  MoveL 3161 to (509.6, 500.88, 6.4) mm, rotated rx 0 ry 90 rz 0 deg; joints [-11.904, -26.782, 109.906, -15.94, -82.523, 51.112]
  Call Extruder(0.254)
  MoveL 3162 to (509.6, 509.6, 6.4) mm, rotated rx 0 ry 90 rz 0 deg; joints [-12.688, -26.745, 109.678, -16.738, -82.366, 51.259]
  Call Extruder(0.559)
  MoveL 3163 to (490.4, 509.6, 6.4) mm, rotated rx 0 ry 90 rz 0 deg; joints [-13.088, -27.092, 111.961, -17.074, -84.231, 50.733]
  MoveL 3164 to (490.4, 490.4, 6.4) mm, rotated rx 0 ry 90 rz 0 deg; joints [-11.303, -27.159, 112.45, -15.27, -84.594, 50.467]
  Call Extruder(0.167)
  MoveL 3165 to (496.12, 490.4, 6.4) mm, rotated rx 0 ry 90 rz 0 deg; joints [-11.197, -27.066, 111.773, -15.179, -84.029, 50.612]
  Call Extruder(0.055)
  MoveL 3166 to (496.12, 492.3, 6.4) mm, rotated rx 0 ry 90 rz 0 deg; joints [-11.373, -27.06, 111.728, -15.356, -83.995, 50.638]
  Call Extruder(0.073)
  MoveL 3167 to (498.63, 492.29, 6.4) mm, rotated rx 0 ry 90 rz 0 deg; joints [-11.326, -27.017, 111.43, -15.316, -83.748, 50.702]
  Call Extruder(0.045)
  MoveL 3168 to (498.63, 490.75, 6.4) mm, rotated rx 0 ry 90 rz 0 deg; joints [-11.183, -27.022, 111.466, -15.172, -83.775, 50.68]
  Call Extruder(0.010)
  MoveL 3169 to (498.63, 490.4, 6.4) mm, rotated rx 0 ry 90 rz 0 deg; joints [-11.151, -27.023, 111.474, -15.14, -83.781, 50.675]
  Call Extruder(0.007)
  MoveL 3170 to (498.98, 490.4, 6.4) mm, rotated rx 0 ry 90 rz 0 deg; joints [-11.145, -27.017, 111.433, -15.134, -83.746, 50.684]
  Call Extruder(0.044)
  MoveL 3171 to (500.51, 490.4, 6.4) mm, rotated rx 0 ry 90 rz 0 deg; joints [-11.117, -26.99, 111.251, -15.111, -83.596, 50.722]
  Call Extruder(0.045)
  MoveL 3172 to (500.51, 491.94, 6.4) mm, rotated rx 0 ry 90 rz 0 deg; joints [-11.259, -26.985, 111.215, -15.255, -83.569, 50.744]
  Call Extruder(0.010)
  MoveL 3173 to (500.51, 492.29, 6.4) mm, rotated rx 0 ry 90 rz 0 deg; joints [-11.291, -26.984, 111.207, -15.287, -83.563, 50.749]
  Call Extruder(0.007)
  MoveL 3174 to (500.86, 492.29, 6.4) mm, rotated rx 0 ry 90 rz 0 deg; joints [-11.285, -26.978, 111.165, -15.282, -83.529, 50.758]
  Call Extruder(0.063)
  MoveL 3175 to (503.03, 492.3, 6.4) mm, rotated rx 0 ry 90 rz 0 deg; joints [-11.245, -26.939, 110.906, -15.249, -83.315, 50.812]
  Call Extruder(0.055)
  MoveL 3176 to (503.03, 490.4, 6.4) mm, rotated rx 0 ry 90 rz 0 deg; joints [-11.072, -26.946, 110.95, -15.073, -83.347, 50.785]
  Call Extruder(0.191)
  MoveL 3177 to (509.6, 490.4, 6.4) mm, rotated rx 0 ry 90 rz 0 deg; joints [-10.955, -26.823, 110.161, -14.976, -82.7, 50.946]
  Call Extruder(0.233)
  MoveL 3178 to (509.6, 498.4, 6.4) mm, rotated rx 0 ry 90 rz 0 deg; joints [-11.68, -26.793, 109.969, -15.712, -82.566, 51.072]
  Call Extruder(0.056)
  MoveL 3179 to (507.66, 498.4, 6.4) mm, rotated rx 0 ry 90 rz 0 deg; joints [-11.716, -26.83, 110.202, -15.742, -82.756, 51.023]
  Set speed (120.0 mm/s)
  MoveL 3180 to (507.66, 498.8, 6.4) mm, rotated rx 0 ry 90 rz 0 deg; joints [-11.752, -26.828, 110.192, -15.779, -82.749, 51.029]
  Set speed (1000.0 mm/s)
  MoveL 3181 to (506.96, 498.8, 6.4) mm, rotated rx 0 ry 90 rz 0 deg; joints [-11.766, -26.842, 110.276, -15.79, -82.818, 51.011]
  Set speed (1000.0 mm/s)
  MoveL 3182 to (490.68, 490.68, 6.4) mm, rotated rx 0 ry 90 rz 0 deg; joints [-11.324, -27.154, 112.411, -15.292, -84.562, 50.478]
  Set speed (1000.0 mm/s)
  MoveL 3183 to (490.68, 490.68, 6.5) mm, rotated rx 0 ry 90 rz 0 deg; joints [-11.324, -27.165, 112.416, -15.292, -84.557, 50.479]
  Set speed (30.0 mm/s)
  Call Extruder(0.767)
  MoveL 3184 to (509.32, 509.32, 6.5) mm, rotated rx 0 ry 90 rz 0 deg; joints [-12.669, -26.762, 109.724, -16.717, -82.394, 51.248]
  MoveL 3185 to (509.44, 509.44, 6.5) mm, rotated rx 0 ry 90 rz 0 deg; joints [-12.677, -26.76, 109.706, -16.726, -82.38, 51.253]
  Set speed (120.0 mm/s)
  MoveL 3186 to (508.74, 501.16, 6.5) mm, rotated rx 0 ry 90 rz 0 deg; joints [-11.945, -26.809, 110.008, -15.979, -82.598, 51.096]
  Set speed (30.0 mm/s)
  Call Extruder(0.336)
  MoveL 3187 to (500.58, 509.32, 6.5) mm, rotated rx 0 ry 90 rz 0 deg; joints [-12.847, -26.928, 110.77, -16.865, -83.242, 51.012]
  Set speed (120.0 mm/s)
  MoveL 3188 to (499.42, 509.32, 6.5) mm, rotated rx 0 ry 90 rz 0 deg; joints [-12.872, -26.949, 110.907, -16.885, -83.355, 50.98]
  Set speed (30.0 mm/s)
  Call Extruder(0.360)
  MoveL 3189 to (490.68, 500.58, 6.5) mm, rotated rx 0 ry 90 rz 0 deg; joints [-12.247, -27.132, 112.172, -16.224, -84.375, 50.612]
  Set speed (120.0 mm/s)
  MoveL 3190 to (490.68, 499.42, 6.5) mm, rotated rx 0 ry 90 rz 0 deg; joints [-12.139, -27.136, 112.202, -16.115, -84.397, 50.596]
  Set speed (30.0 mm/s)
  Call Extruder(0.282)
  MoveL 3191 to (497.52, 492.57, 6.5) mm, rotated rx 0 ry 90 rz 0 deg; joints [-11.372, -27.045, 111.56, -15.36, -83.847, 50.679]
  MoveL 3192 to (497.65, 492.45, 6.5) mm, rotated rx 0 ry 90 rz 0 deg; joints [-11.359, -27.044, 111.549, -15.347, -83.837, 50.68]
  Set speed (120.0 mm/s)
  MoveL 3193 to (498.97, 491.13, 6.5) mm, rotated rx 0 ry 90 rz 0 deg; joints [-11.212, -27.025, 111.422, -15.202, -83.73, 50.695]
  Set speed (30.0 mm/s)
  Call Extruder(0.018)
  MoveL 3194 to (499.42, 490.68, 6.5) mm, rotated rx 0 ry 90 rz 0 deg; joints [-11.163, -27.019, 111.38, -15.154, -83.693, 50.7]
  Set speed (120.0 mm/s)
  MoveL 3195 to (500.42, 492.32, 6.5) mm, rotated rx 0 ry 90 rz 0 deg; joints [-11.296, -26.996, 111.222, -15.292, -83.567, 50.749]
  Set speed (1000.0 mm/s)
  MoveL 3196 to (502.47, 492.57, 6.5) mm, rotated rx 0 ry 90 rz 0 deg; joints [-11.281, -26.958, 110.97, -15.283, -83.36, 50.804]
  Set speed (30.0 mm/s)
  Call Extruder(0.228)
  MoveL 3197 to (508.02, 498.12, 6.5) mm, rotated rx 0 ry 90 rz 0 deg; joints [-11.684, -26.835, 110.171, -15.711, -82.721, 51.029]
  MoveL 3198 to (508.14, 498.24, 6.5) mm, rotated rx 0 ry 90 rz 0 deg; joints [-11.693, -26.832, 110.153, -15.72, -82.707, 51.034]
  Set speed (120.0 mm/s)
  MoveL 3199 to (509.32, 490.68, 6.5) mm, rotated rx 0 ry 90 rz 0 deg; joints [-10.985, -26.838, 110.194, -15.006, -82.718, 50.945]
  Set speed (30.0 mm/s)
  Call Extruder(0.767)
  MoveL 3200 to (490.68, 509.32, 6.5) mm, rotated rx 0 ry 90 rz 0 deg; joints [-13.056, -27.1, 111.941, -17.043, -84.205, 50.738]
  MoveL 3201 to (490.56, 509.44, 6.5) mm, rotated rx 0 ry 90 rz 0 deg; joints [-13.07, -27.101, 111.952, -17.057, -84.214, 50.736]
  Set speed (120.0 mm/s)
  MoveL 3202 to (507.59, 498.33, 6.5) mm, rotated rx 0 ry 90 rz 0 deg; joints [-11.711, -26.842, 110.217, -15.737, -82.759, 51.021]
  Set speed (1000.0 mm/s)
  MoveL 3203 to (507.66, 498.4, 6.5) mm, rotated rx 0 ry 90 rz 0 deg; joints [-11.716, -26.84, 110.207, -15.742, -82.751, 51.024]
  Set speed (15.0 mm/s)
  Call Extruder(0.072)
  MoveL 3204 to (507.66, 500.88, 6.5) mm, rotated rx 0 ry 90 rz 0 deg; joints [-11.941, -26.83, 110.145, -15.97, -82.708, 51.064]
  Call Extruder(0.056)
  MoveL 3205 to (509.6, 500.88, 6.5) mm, rotated rx 0 ry 90 rz 0 deg; joints [-11.904, -26.793, 109.911, -15.94, -82.518, 51.114]
  Call Extruder(0.254)
  MoveL 3206 to (509.6, 509.6, 6.5) mm, rotated rx 0 ry 90 rz 0 deg; joints [-12.688, -26.756, 109.683, -16.738, -82.361, 51.26]
  Call Extruder(0.559)
  MoveL 3207 to (490.4, 509.6, 6.5) mm, rotated rx 0 ry 90 rz 0 deg; joints [-13.088, -27.103, 111.966, -17.074, -84.226, 50.734]
  MoveL 3208 to (490.4, 490.4, 6.5) mm, rotated rx 0 ry 90 rz 0 deg; joints [-11.303, -27.17, 112.456, -15.27, -84.589, 50.468]
  Call Extruder(0.168)
  MoveL 3209 to (496.18, 490.4, 6.5) mm, rotated rx 0 ry 90 rz 0 deg; joints [-11.196, -27.076, 111.772, -15.178, -84.018, 50.615]
  Call Extruder(0.045)
  MoveL 3210 to (496.18, 491.94, 6.5) mm, rotated rx 0 ry 90 rz 0 deg; joints [-11.339, -27.07, 111.735, -15.323, -83.991, 50.636]
  Call Extruder(0.010)
  MoveL 3211 to (496.18, 492.3, 6.5) mm, rotated rx 0 ry 90 rz 0 deg; joints [-11.372, -27.069, 111.727, -15.355, -83.985, 50.641]
  Call Extruder(0.007)
  MoveL 3212 to (496.53, 492.3, 6.5) mm, rotated rx 0 ry 90 rz 0 deg; joints [-11.365, -27.063, 111.685, -15.35, -83.95, 50.65]
  Call Extruder(0.063)
  MoveL 3213 to (498.69, 492.29, 6.5) mm, rotated rx 0 ry 90 rz 0 deg; joints [-11.325, -27.026, 111.428, -15.316, -83.737, 50.705]
  Call Extruder(0.045)
  MoveL 3214 to (498.69, 490.75, 6.5) mm, rotated rx 0 ry 90 rz 0 deg; joints [-11.182, -27.032, 111.465, -15.172, -83.764, 50.683]
  Call Extruder(0.010)
  MoveL 3215 to (498.69, 490.4, 6.5) mm, rotated rx 0 ry 90 rz 0 deg; joints [-11.15, -27.033, 111.473, -15.139, -83.77, 50.678]
  Call Extruder(0.007)
  MoveL 3216 to (499.04, 490.4, 6.5) mm, rotated rx 0 ry 90 rz 0 deg; joints [-11.144, -27.027, 111.431, -15.133, -83.735, 50.687]
  Call Extruder(0.041)
  MoveL 3217 to (500.45, 490.4, 6.5) mm, rotated rx 0 ry 90 rz 0 deg; joints [-11.118, -27.002, 111.264, -15.112, -83.597, 50.722]
  Call Extruder(0.045)
  MoveL 3218 to (500.45, 491.94, 6.5) mm, rotated rx 0 ry 90 rz 0 deg; joints [-11.26, -26.997, 111.227, -15.256, -83.57, 50.744]
  Call Extruder(0.010)
  MoveL 3219 to (500.45, 492.29, 6.5) mm, rotated rx 0 ry 90 rz 0 deg; joints [-11.293, -26.996, 111.219, -15.288, -83.564, 50.749]
  Call Extruder(0.007)
  MoveL 3220 to (500.8, 492.29, 6.5) mm, rotated rx 0 ry 90 rz 0 deg; joints [-11.286, -26.989, 111.177, -15.283, -83.53, 50.758]
  Call Extruder(0.063)
  MoveL 3221 to (502.96, 492.3, 6.5) mm, rotated rx 0 ry 90 rz 0 deg; joints [-11.247, -26.951, 110.918, -15.25, -83.316, 50.812]
  Call Extruder(0.055)
  MoveL 3222 to (502.97, 490.4, 6.5) mm, rotated rx 0 ry 90 rz 0 deg; joints [-11.073, -26.957, 110.963, -15.074, -83.348, 50.784]
  Call Extruder(0.193)
  MoveL 3223 to (509.6, 490.4, 6.5) mm, rotated rx 0 ry 90 rz 0 deg; joints [-10.955, -26.834, 110.167, -14.977, -82.695, 50.948]
  Call Extruder(0.233)
  MoveL 3224 to (509.6, 498.4, 6.5) mm, rotated rx 0 ry 90 rz 0 deg; joints [-11.68, -26.803, 109.974, -15.712, -82.561, 51.074]
  Call Extruder(0.056)
  MoveL 3225 to (507.66, 498.4, 6.5) mm, rotated rx 0 ry 90 rz 0 deg; joints [-11.716, -26.84, 110.207, -15.742, -82.751, 51.024]
  Set speed (120.0 mm/s)
  MoveL 3226 to (507.66, 498.8, 6.5) mm, rotated rx 0 ry 90 rz 0 deg; joints [-11.752, -26.839, 110.197, -15.779, -82.744, 51.03]
  Set speed (1000.0 mm/s)
  MoveL 3227 to (506.96, 498.8, 6.5) mm, rotated rx 0 ry 90 rz 0 deg; joints [-11.766, -26.852, 110.281, -15.79, -82.813, 51.013]
  Set speed (1000.0 mm/s)
  MoveL 3228 to (490.68, 490.68, 6.5) mm, rotated rx 0 ry 90 rz 0 deg; joints [-11.324, -27.165, 112.416, -15.292, -84.557, 50.479]
  Set speed (1000.0 mm/s)
  MoveL 3229 to (490.68, 490.68, 6.6) mm, rotated rx 0 ry 90 rz 0 deg; joints [-11.324, -27.175, 112.421, -15.292, -84.551, 50.481]
  Set speed (30.0 mm/s)
  Call Extruder(0.767)
  MoveL 3230 to (509.32, 509.32, 6.6) mm, rotated rx 0 ry 90 rz 0 deg; joints [-12.669, -26.773, 109.729, -16.717, -82.389, 51.25]
  MoveL 3231 to (509.44, 509.44, 6.6) mm, rotated rx 0 ry 90 rz 0 deg; joints [-12.677, -26.77, 109.711, -16.726, -82.375, 51.255]
  Set speed (120.0 mm/s)
  MoveL 3232 to (508.74, 501.16, 6.6) mm, rotated rx 0 ry 90 rz 0 deg; joints [-11.945, -26.819, 110.013, -15.979, -82.592, 51.098]
  Set speed (30.0 mm/s)
  Call Extruder(0.336)
  MoveL 3233 to (500.58, 509.32, 6.6) mm, rotated rx 0 ry 90 rz 0 deg; joints [-12.847, -26.938, 110.775, -16.865, -83.237, 51.013]
  Set speed (120.0 mm/s)
  MoveL 3234 to (499.42, 509.32, 6.6) mm, rotated rx 0 ry 90 rz 0 deg; joints [-12.872, -26.959, 110.913, -16.886, -83.35, 50.982]
  Set speed (30.0 mm/s)
  Call Extruder(0.360)
  MoveL 3235 to (490.68, 500.58, 6.6) mm, rotated rx 0 ry 90 rz 0 deg; joints [-12.247, -27.142, 112.178, -16.224, -84.37, 50.614]
  Set speed (120.0 mm/s)
  MoveL 3236 to (490.68, 499.42, 6.6) mm, rotated rx 0 ry 90 rz 0 deg; joints [-12.139, -27.146, 112.207, -16.115, -84.392, 50.598]
  Set speed (30.0 mm/s)
  Call Extruder(0.282)
  MoveL 3237 to (497.52, 492.57, 6.6) mm, rotated rx 0 ry 90 rz 0 deg; joints [-11.372, -27.056, 111.566, -15.36, -83.842, 50.68]
  MoveL 3238 to (497.65, 492.45, 6.6) mm, rotated rx 0 ry 90 rz 0 deg; joints [-11.359, -27.054, 111.554, -15.347, -83.832, 50.682]
  Set speed (120.0 mm/s)
  MoveL 3239 to (499.03, 491.07, 6.6) mm, rotated rx 0 ry 90 rz 0 deg; joints [-11.205, -27.035, 111.422, -15.196, -83.72, 50.697]
  Set speed (30.0 mm/s)
  Call Extruder(0.016)
  MoveL 3240 to (499.42, 490.68, 6.6) mm, rotated rx 0 ry 90 rz 0 deg; joints [-11.163, -27.03, 111.385, -15.154, -83.688, 50.702]
  Set speed (120.0 mm/s)
  MoveL 3241 to (500.36, 492.32, 6.6) mm, rotated rx 0 ry 90 rz 0 deg; joints [-11.297, -27.008, 111.234, -15.293, -83.568, 50.748]
  Set speed (1000.0 mm/s)
  MoveL 3242 to (502.47, 492.57, 6.6) mm, rotated rx 0 ry 90 rz 0 deg; joints [-11.281, -26.969, 110.976, -15.284, -83.355, 50.805]
  Set speed (30.0 mm/s)
  Call Extruder(0.228)
  MoveL 3243 to (508.02, 498.12, 6.6) mm, rotated rx 0 ry 90 rz 0 deg; joints [-11.684, -26.845, 110.176, -15.711, -82.716, 51.03]
  MoveL 3244 to (508.14, 498.24, 6.6) mm, rotated rx 0 ry 90 rz 0 deg; joints [-11.693, -26.842, 110.159, -15.72, -82.702, 51.035]
  Set speed (120.0 mm/s)
  MoveL 3245 to (509.32, 490.68, 6.6) mm, rotated rx 0 ry 90 rz 0 deg; joints [-10.985, -26.849, 110.199, -15.006, -82.713, 50.946]
  Set speed (30.0 mm/s)
  Call Extruder(0.767)
  MoveL 3246 to (490.68, 509.32, 6.6) mm, rotated rx 0 ry 90 rz 0 deg; joints [-13.056, -27.11, 111.947, -17.043, -84.2, 50.74]
  MoveL 3247 to (490.56, 509.44, 6.6) mm, rotated rx 0 ry 90 rz 0 deg; joints [-13.07, -27.112, 111.958, -17.057, -84.209, 50.738]
  Set speed (120.0 mm/s)
  MoveL 3248 to (507.59, 498.33, 6.6) mm, rotated rx 0 ry 90 rz 0 deg; joints [-11.711, -26.852, 110.223, -15.737, -82.754, 51.023]
  Set speed (1000.0 mm/s)
  MoveL 3249 to (507.66, 498.4, 6.6) mm, rotated rx 0 ry 90 rz 0 deg; joints [-11.716, -26.851, 110.212, -15.742, -82.746, 51.026]
  Set speed (15.0 mm/s)
  Call Extruder(0.072)
  MoveL 3250 to (507.66, 500.88, 6.6) mm, rotated rx 0 ry 90 rz 0 deg; joints [-11.941, -26.841, 110.15, -15.97, -82.703, 51.065]
  Call Extruder(0.056)
  MoveL 3251 to (509.6, 500.88, 6.6) mm, rotated rx 0 ry 90 rz 0 deg; joints [-11.904, -26.803, 109.917, -15.94, -82.513, 51.115]
  Call Extruder(0.254)
  MoveL 3252 to (509.6, 509.6, 6.6) mm, rotated rx 0 ry 90 rz 0 deg; joints [-12.688, -26.766, 109.688, -16.738, -82.356, 51.262]
  Call Extruder(0.559)
  MoveL 3253 to (490.4, 509.6, 6.6) mm, rotated rx 0 ry 90 rz 0 deg; joints [-13.088, -27.114, 111.972, -17.074, -84.221, 50.736]
  MoveL 3254 to (490.4, 490.4, 6.6) mm, rotated rx 0 ry 90 rz 0 deg; joints [-11.303, -27.181, 112.461, -15.27, -84.584, 50.47]
  Call Extruder(0.170)
  MoveL 3255 to (496.23, 490.4, 6.6) mm, rotated rx 0 ry 90 rz 0 deg; joints [-11.195, -27.085, 111.771, -15.177, -84.007, 50.618]
  Call Extruder(0.055)
  MoveL 3256 to (496.24, 492.3, 6.6) mm, rotated rx 0 ry 90 rz 0 deg; joints [-11.371, -27.079, 111.725, -15.355, -83.974, 50.644]
  Call Extruder(0.073)
  MoveL 3257 to (498.75, 492.29, 6.6) mm, rotated rx 0 ry 90 rz 0 deg; joints [-11.324, -27.036, 111.426, -15.315, -83.726, 50.708]
  Call Extruder(0.045)
  MoveL 3258 to (498.75, 490.75, 6.6) mm, rotated rx 0 ry 90 rz 0 deg; joints [-11.181, -27.041, 111.463, -15.171, -83.753, 50.686]
  Call Extruder(0.010)
  MoveL 3259 to (498.75, 490.4, 6.6) mm, rotated rx 0 ry 90 rz 0 deg; joints [-11.149, -27.042, 111.471, -15.138, -83.759, 50.681]
  Call Extruder(0.007)
  MoveL 3260 to (499.1, 490.4, 6.6) mm, rotated rx 0 ry 90 rz 0 deg; joints [-11.143, -27.036, 111.429, -15.133, -83.724, 50.69]
  Call Extruder(0.037)
  MoveL 3261 to (500.39, 490.4, 6.6) mm, rotated rx 0 ry 90 rz 0 deg; joints [-11.119, -27.014, 111.276, -15.113, -83.597, 50.722]
  Call Extruder(0.045)
  MoveL 3262 to (500.38, 491.94, 6.6) mm, rotated rx 0 ry 90 rz 0 deg; joints [-11.261, -27.008, 111.24, -15.257, -83.571, 50.744]
  Call Extruder(0.010)
  MoveL 3263 to (500.39, 492.29, 6.6) mm, rotated rx 0 ry 90 rz 0 deg; joints [-11.294, -27.007, 111.232, -15.29, -83.565, 50.749]
  Call Extruder(0.007)
  MoveL 3264 to (500.73, 492.29, 6.6) mm, rotated rx 0 ry 90 rz 0 deg; joints [-11.287, -27.001, 111.19, -15.284, -83.531, 50.758]
  Call Extruder(0.063)
  MoveL 3265 to (502.9, 492.3, 6.6) mm, rotated rx 0 ry 90 rz 0 deg; joints [-11.248, -26.962, 110.931, -15.251, -83.318, 50.812]
  Call Extruder(0.055)
  MoveL 3266 to (502.9, 490.4, 6.6) mm, rotated rx 0 ry 90 rz 0 deg; joints [-11.074, -26.969, 110.976, -15.075, -83.349, 50.784]
  Call Extruder(0.195)
  MoveL 3267 to (509.6, 490.4, 6.6) mm, rotated rx 0 ry 90 rz 0 deg; joints [-10.955, -26.844, 110.172, -14.977, -82.69, 50.949]
  Call Extruder(0.233)
  MoveL 3268 to (509.6, 498.4, 6.6) mm, rotated rx 0 ry 90 rz 0 deg; joints [-11.68, -26.813, 109.979, -15.713, -82.556, 51.075]
  Call Extruder(0.056)
  MoveL 3269 to (507.66, 498.4, 6.6) mm, rotated rx 0 ry 90 rz 0 deg; joints [-11.716, -26.851, 110.212, -15.742, -82.746, 51.026]
  Set speed (120.0 mm/s)
  MoveL 3270 to (507.66, 498.8, 6.6) mm, rotated rx 0 ry 90 rz 0 deg; joints [-11.752, -26.849, 110.202, -15.779, -82.739, 51.032]
  Set speed (1000.0 mm/s)
  MoveL 3271 to (506.96, 498.8, 6.6) mm, rotated rx 0 ry 90 rz 0 deg; joints [-11.765, -26.863, 110.287, -15.79, -82.808, 51.014]
  Set speed (1000.0 mm/s)
  MoveL 3272 to (490.68, 490.68, 6.6) mm, rotated rx 0 ry 90 rz 0 deg; joints [-11.324, -27.175, 112.421, -15.292, -84.551, 50.481]
  Set speed (1000.0 mm/s)
  MoveL 3273 to (490.68, 490.68, 6.7) mm, rotated rx 0 ry 90 rz 0 deg; joints [-11.324, -27.186, 112.427, -15.292, -84.546, 50.482]
  Set speed (30.0 mm/s)
  Call Extruder(0.767)
  MoveL 3274 to (509.32, 509.32, 6.7) mm, rotated rx 0 ry 90 rz 0 deg; joints [-12.669, -26.783, 109.735, -16.717, -82.384, 51.251]
  MoveL 3275 to (509.44, 509.44, 6.7) mm, rotated rx 0 ry 90 rz 0 deg; joints [-12.677, -26.78, 109.717, -16.727, -82.37, 51.257]
  Set speed (120.0 mm/s)
  MoveL 3276 to (508.74, 501.16, 6.7) mm, rotated rx 0 ry 90 rz 0 deg; joints [-11.945, -26.829, 110.018, -15.979, -82.587, 51.099]
  Set speed (30.0 mm/s)
  Call Extruder(0.336)
  MoveL 3277 to (500.58, 509.32, 6.7) mm, rotated rx 0 ry 90 rz 0 deg; joints [-12.847, -26.949, 110.78, -16.866, -83.232, 51.015]
  Set speed (120.0 mm/s)
  MoveL 3278 to (499.42, 509.32, 6.7) mm, rotated rx 0 ry 90 rz 0 deg; joints [-12.872, -26.97, 110.918, -16.886, -83.345, 50.983]
  Set speed (30.0 mm/s)
  Call Extruder(0.360)
  MoveL 3279 to (490.68, 500.58, 6.7) mm, rotated rx 0 ry 90 rz 0 deg; joints [-12.247, -27.153, 112.183, -16.224, -84.365, 50.615]
  Set speed (120.0 mm/s)
  MoveL 3280 to (490.68, 499.42, 6.7) mm, rotated rx 0 ry 90 rz 0 deg; joints [-12.139, -27.157, 112.213, -16.115, -84.387, 50.599]
  Set speed (30.0 mm/s)
  Call Extruder(0.282)
  MoveL 3281 to (497.52, 492.57, 6.7) mm, rotated rx 0 ry 90 rz 0 deg; joints [-11.372, -27.067, 111.571, -15.36, -83.837, 50.682]
  MoveL 3282 to (497.65, 492.45, 6.7) mm, rotated rx 0 ry 90 rz 0 deg; joints [-11.359, -27.065, 111.559, -15.347, -83.827, 50.683]
  Set speed (120.0 mm/s)
  MoveL 3283 to (499.09, 491.01, 6.7) mm, rotated rx 0 ry 90 rz 0 deg; joints [-11.199, -27.045, 111.422, -15.19, -83.71, 50.699]
  Set speed (30.0 mm/s)
  Call Extruder(0.013)
  MoveL 3284 to (499.42, 490.68, 6.7) mm, rotated rx 0 ry 90 rz 0 deg; joints [-11.163, -27.04, 111.39, -15.154, -83.683, 50.703]
  Set speed (120.0 mm/s)
  MoveL 3285 to (500.3, 492.32, 6.7) mm, rotated rx 0 ry 90 rz 0 deg; joints [-11.298, -27.019, 111.247, -15.294, -83.569, 50.748]
  Set speed (1000.0 mm/s)
  MoveL 3286 to (502.47, 492.57, 6.7) mm, rotated rx 0 ry 90 rz 0 deg; joints [-11.281, -26.979, 110.981, -15.284, -83.35, 50.807]
  Set speed (30.0 mm/s)
  Call Extruder(0.228)
  MoveL 3287 to (508.02, 498.12, 6.7) mm, rotated rx 0 ry 90 rz 0 deg; joints [-11.684, -26.856, 110.182, -15.711, -82.711, 51.032]
  MoveL 3288 to (508.14, 498.24, 6.7) mm, rotated rx 0 ry 90 rz 0 deg; joints [-11.693, -26.853, 110.164, -15.721, -82.697, 51.037]
  Set speed (120.0 mm/s)
  MoveL 3289 to (509.32, 490.68, 6.7) mm, rotated rx 0 ry 90 rz 0 deg; joints [-10.985, -26.859, 110.204, -15.007, -82.708, 50.948]
  Set speed (30.0 mm/s)
  Call Extruder(0.767)
  MoveL 3290 to (490.68, 509.32, 6.7) mm, rotated rx 0 ry 90 rz 0 deg; joints [-13.056, -27.121, 111.952, -17.043, -84.195, 50.741]
  MoveL 3291 to (490.56, 509.44, 6.7) mm, rotated rx 0 ry 90 rz 0 deg; joints [-13.07, -27.122, 111.963, -17.057, -84.204, 50.74]
  Set speed (120.0 mm/s)
  MoveL 3292 to (507.59, 498.33, 6.7) mm, rotated rx 0 ry 90 rz 0 deg; joints [-11.711, -26.863, 110.228, -15.737, -82.749, 51.024]
  Set speed (1000.0 mm/s)
  MoveL 3293 to (507.66, 498.4, 6.7) mm, rotated rx 0 ry 90 rz 0 deg; joints [-11.716, -26.861, 110.218, -15.742, -82.741, 51.027]
  Set speed (15.0 mm/s)
  Call Extruder(0.072)
  MoveL 3294 to (507.66, 500.88, 6.7) mm, rotated rx 0 ry 90 rz 0 deg; joints [-11.94, -26.851, 110.155, -15.971, -82.698, 51.067]
  Call Extruder(0.056)
  MoveL 3295 to (509.6, 500.88, 6.7) mm, rotated rx 0 ry 90 rz 0 deg; joints [-11.904, -26.814, 109.922, -15.94, -82.508, 51.117]
  Call Extruder(0.254)
  MoveL 3296 to (509.6, 509.6, 6.7) mm, rotated rx 0 ry 90 rz 0 deg; joints [-12.688, -26.777, 109.693, -16.739, -82.351, 51.263]
  Call Extruder(0.559)
  MoveL 3297 to (490.4, 509.6, 6.7) mm, rotated rx 0 ry 90 rz 0 deg; joints [-13.088, -27.124, 111.977, -17.075, -84.216, 50.738]
  MoveL 3298 to (490.4, 490.4, 6.7) mm, rotated rx 0 ry 90 rz 0 deg; joints [-11.303, -27.191, 112.466, -15.27, -84.579, 50.471]
  Call Extruder(0.171)
  MoveL 3299 to (496.29, 490.4, 6.7) mm, rotated rx 0 ry 90 rz 0 deg; joints [-11.194, -27.095, 111.769, -15.176, -83.997, 50.621]
  Call Extruder(0.045)
  MoveL 3300 to (496.29, 491.95, 6.7) mm, rotated rx 0 ry 90 rz 0 deg; joints [-11.337, -27.09, 111.732, -15.321, -83.97, 50.642]
  Call Extruder(0.010)
  MoveL 3301 to (496.29, 492.3, 6.7) mm, rotated rx 0 ry 90 rz 0 deg; joints [-11.37, -27.089, 111.724, -15.354, -83.964, 50.647]
  Call Extruder(0.007)
  MoveL 3302 to (496.64, 492.3, 6.7) mm, rotated rx 0 ry 90 rz 0 deg; joints [-11.363, -27.083, 111.683, -15.348, -83.929, 50.656]
  Call Extruder(0.063)
  MoveL 3303 to (498.81, 492.29, 6.7) mm, rotated rx 0 ry 90 rz 0 deg; joints [-11.323, -27.045, 111.424, -15.314, -83.715, 50.711]
  Call Extruder(0.045)
  MoveL 3304 to (498.81, 490.75, 6.7) mm, rotated rx 0 ry 90 rz 0 deg; joints [-11.18, -27.051, 111.461, -15.17, -83.742, 50.689]
  Call Extruder(0.010)
  MoveL 3305 to (498.81, 490.4, 6.7) mm, rotated rx 0 ry 90 rz 0 deg; joints [-11.148, -27.052, 111.469, -15.137, -83.748, 50.684]
  Call Extruder(0.007)
  MoveL 3306 to (499.16, 490.4, 6.7) mm, rotated rx 0 ry 90 rz 0 deg; joints [-11.141, -27.046, 111.427, -15.132, -83.713, 50.693]
  Call Extruder(0.034)
  MoveL 3307 to (500.33, 490.4, 6.7) mm, rotated rx 0 ry 90 rz 0 deg; joints [-11.12, -27.025, 111.289, -15.114, -83.598, 50.722]
  Call Extruder(0.045)
  MoveL 3308 to (500.32, 491.94, 6.7) mm, rotated rx 0 ry 90 rz 0 deg; joints [-11.263, -27.02, 111.253, -15.258, -83.572, 50.744]
  Call Extruder(0.010)
  MoveL 3309 to (500.32, 492.29, 6.7) mm, rotated rx 0 ry 90 rz 0 deg; joints [-11.295, -27.019, 111.244, -15.291, -83.566, 50.749]
  Call Extruder(0.007)
  MoveL 3310 to (500.67, 492.29, 6.7) mm, rotated rx 0 ry 90 rz 0 deg; joints [-11.288, -27.013, 111.202, -15.285, -83.532, 50.757]
  Call Extruder(0.063)
  MoveL 3311 to (502.84, 492.3, 6.7) mm, rotated rx 0 ry 90 rz 0 deg; joints [-11.249, -26.974, 110.944, -15.252, -83.319, 50.812]
  Call Extruder(0.055)
  MoveL 3312 to (502.84, 490.4, 6.7) mm, rotated rx 0 ry 90 rz 0 deg; joints [-11.075, -26.981, 110.989, -15.076, -83.351, 50.784]
  Call Extruder(0.197)
  MoveL 3313 to (509.6, 490.4, 6.7) mm, rotated rx 0 ry 90 rz 0 deg; joints [-10.955, -26.855, 110.177, -14.977, -82.685, 50.95]
  Call Extruder(0.233)
  MoveL 3314 to (509.6, 498.4, 6.7) mm, rotated rx 0 ry 90 rz 0 deg; joints [-11.679, -26.824, 109.984, -15.713, -82.551, 51.076]
  Call Extruder(0.056)
  MoveL 3315 to (507.66, 498.4, 6.7) mm, rotated rx 0 ry 90 rz 0 deg; joints [-11.716, -26.861, 110.218, -15.742, -82.741, 51.027]
  Set speed (120.0 mm/s)
  MoveL 3316 to (507.66, 498.8, 6.7) mm, rotated rx 0 ry 90 rz 0 deg; joints [-11.752, -26.86, 110.208, -15.779, -82.734, 51.033]
  Set speed (1000.0 mm/s)
  MoveL 3317 to (506.96, 498.8, 6.7) mm, rotated rx 0 ry 90 rz 0 deg; joints [-11.765, -26.873, 110.292, -15.79, -82.803, 51.015]
  Set speed (1000.0 mm/s)
  MoveL 3318 to (490.68, 490.68, 6.7) mm, rotated rx 0 ry 90 rz 0 deg; joints [-11.324, -27.186, 112.427, -15.292, -84.546, 50.482]
  Set speed (1000.0 mm/s)
  MoveL 3319 to (490.68, 490.68, 6.8) mm, rotated rx 0 ry 90 rz 0 deg; joints [-11.324, -27.197, 112.432, -15.292, -84.541, 50.483]
  Set speed (30.0 mm/s)
  Call Extruder(0.767)
  MoveL 3320 to (509.32, 509.32, 6.8) mm, rotated rx 0 ry 90 rz 0 deg; joints [-12.669, -26.794, 109.74, -16.718, -82.379, 51.253]
  MoveL 3321 to (509.44, 509.44, 6.8) mm, rotated rx 0 ry 90 rz 0 deg; joints [-12.677, -26.791, 109.722, -16.727, -82.365, 51.258]
  Set speed (120.0 mm/s)
  MoveL 3322 to (508.74, 501.16, 6.8) mm, rotated rx 0 ry 90 rz 0 deg; joints [-11.945, -26.84, 110.023, -15.979, -82.582, 51.101]
  Set speed (30.0 mm/s)
  Call Extruder(0.336)
  MoveL 3323 to (500.58, 509.32, 6.8) mm, rotated rx 0 ry 90 rz 0 deg; joints [-12.847, -26.96, 110.785, -16.866, -83.227, 51.016]
  Set speed (120.0 mm/s)
  MoveL 3324 to (499.42, 509.32, 6.8) mm, rotated rx 0 ry 90 rz 0 deg; joints [-12.872, -26.98, 110.923, -16.886, -83.34, 50.985]
  Set speed (30.0 mm/s)
  Call Extruder(0.360)
  MoveL 3325 to (490.68, 500.58, 6.8) mm, rotated rx 0 ry 90 rz 0 deg; joints [-12.247, -27.164, 112.188, -16.225, -84.36, 50.617]
  Set speed (120.0 mm/s)
  MoveL 3326 to (490.68, 499.42, 6.8) mm, rotated rx 0 ry 90 rz 0 deg; joints [-12.139, -27.168, 112.218, -16.116, -84.382, 50.6]
  Set speed (30.0 mm/s)
  Call Extruder(0.282)
  MoveL 3327 to (497.53, 492.57, 6.8) mm, rotated rx 0 ry 90 rz 0 deg; joints [-11.372, -27.077, 111.576, -15.361, -83.832, 50.683]
  MoveL 3328 to (497.65, 492.45, 6.8) mm, rotated rx 0 ry 90 rz 0 deg; joints [-11.359, -27.075, 111.564, -15.347, -83.822, 50.685]
  Set speed (120.0 mm/s)
  MoveL 3329 to (502.47, 492.58, 6.8) mm, rotated rx 0 ry 90 rz 0 deg; joints [-11.281, -26.99, 110.986, -15.284, -83.345, 50.808]
  Set speed (30.0 mm/s)
  Call Extruder(0.228)
  MoveL 3330 to (508.01, 498.12, 6.8) mm, rotated rx 0 ry 90 rz 0 deg; joints [-11.684, -26.866, 110.187, -15.711, -82.706, 51.033]
  MoveL 3331 to (508.14, 498.24, 6.8) mm, rotated rx 0 ry 90 rz 0 deg; joints [-11.692, -26.863, 110.169, -15.721, -82.692, 51.038]
  Set speed (120.0 mm/s)
  MoveL 3332 to (509.32, 490.68, 6.8) mm, rotated rx 0 ry 90 rz 0 deg; joints [-10.985, -26.87, 110.21, -15.007, -82.703, 50.949]
  Set speed (30.0 mm/s)
  Call Extruder(0.767)
  MoveL 3333 to (490.68, 509.32, 6.8) mm, rotated rx 0 ry 90 rz 0 deg; joints [-13.056, -27.131, 111.957, -17.043, -84.19, 50.743]
  MoveL 3334 to (490.56, 509.44, 6.8) mm, rotated rx 0 ry 90 rz 0 deg; joints [-13.07, -27.133, 111.968, -17.057, -84.199, 50.741]
  Set speed (120.0 mm/s)
  MoveL 3335 to (507.59, 498.33, 6.8) mm, rotated rx 0 ry 90 rz 0 deg; joints [-11.711, -26.873, 110.233, -15.737, -82.744, 51.025]
  Set speed (1000.0 mm/s)
  MoveL 3336 to (507.66, 498.4, 6.8) mm, rotated rx 0 ry 90 rz 0 deg; joints [-11.716, -26.872, 110.223, -15.743, -82.736, 51.028]
  Set speed (15.0 mm/s)
  Call Extruder(0.072)
  MoveL 3337 to (507.66, 500.88, 6.8) mm, rotated rx 0 ry 90 rz 0 deg; joints [-11.94, -26.862, 110.161, -15.971, -82.693, 51.068]
  Call Extruder(0.056)
  MoveL 3338 to (509.6, 500.88, 6.8) mm, rotated rx 0 ry 90 rz 0 deg; joints [-11.903, -26.824, 109.927, -15.94, -82.503, 51.118]
  Call Extruder(0.254)
  MoveL 3339 to (509.6, 509.6, 6.8) mm, rotated rx 0 ry 90 rz 0 deg; joints [-12.688, -26.787, 109.699, -16.739, -82.347, 51.265]
  Call Extruder(0.559)
  MoveL 3340 to (490.4, 509.6, 6.8) mm, rotated rx 0 ry 90 rz 0 deg; joints [-13.088, -27.135, 111.982, -17.075, -84.211, 50.739]
  MoveL 3341 to (490.4, 490.4, 6.8) mm, rotated rx 0 ry 90 rz 0 deg; joints [-11.303, -27.202, 112.472, -15.27, -84.574, 50.473]
  Call Extruder(0.173)
  MoveL 3342 to (496.34, 490.4, 6.8) mm, rotated rx 0 ry 90 rz 0 deg; joints [-11.193, -27.105, 111.768, -15.176, -83.986, 50.623]
  Call Extruder(0.055)
  MoveL 3343 to (496.35, 492.3, 6.8) mm, rotated rx 0 ry 90 rz 0 deg; joints [-11.368, -27.098, 111.723, -15.353, -83.953, 50.649]
  Call Extruder(0.063)
  MoveL 3344 to (498.52, 492.29, 6.8) mm, rotated rx 0 ry 90 rz 0 deg; joints [-11.328, -27.061, 111.464, -15.319, -83.739, 50.705]
  Call Extruder(0.010)
  MoveL 3345 to (498.87, 492.29, 6.8) mm, rotated rx 0 ry 90 rz 0 deg; joints [-11.322, -27.055, 111.423, -15.313, -83.704, 50.713]
  Call Extruder(0.007)
  MoveL 3346 to (498.87, 491.94, 6.8) mm, rotated rx 0 ry 90 rz 0 deg; joints [-11.289, -27.056, 111.431, -15.281, -83.71, 50.708]
  Call Extruder(0.035)
  MoveL 3347 to (498.87, 490.75, 6.8) mm, rotated rx 0 ry 90 rz 0 deg; joints [-11.179, -27.06, 111.459, -15.169, -83.731, 50.692]
  Call Extruder(0.010)
  MoveL 3348 to (498.87, 490.4, 6.8) mm, rotated rx 0 ry 90 rz 0 deg; joints [-11.147, -27.061, 111.467, -15.137, -83.737, 50.687]
  Call Extruder(0.007)
  MoveL 3349 to (499.22, 490.4, 6.8) mm, rotated rx 0 ry 90 rz 0 deg; joints [-11.14, -27.055, 111.426, -15.131, -83.702, 50.695]
  Call Extruder(0.030)
  MoveL 3350 to (500.26, 490.4, 6.8) mm, rotated rx 0 ry 90 rz 0 deg; joints [-11.121, -27.037, 111.301, -15.115, -83.599, 50.721]
  Call Extruder(0.055)
  MoveL 3351 to (500.26, 492.3, 6.8) mm, rotated rx 0 ry 90 rz 0 deg; joints [-11.296, -27.03, 111.257, -15.292, -83.567, 50.749]
  Call Extruder(0.073)
  MoveL 3352 to (502.77, 492.3, 6.8) mm, rotated rx 0 ry 90 rz 0 deg; joints [-11.25, -26.986, 110.957, -15.253, -83.32, 50.812]
  Call Extruder(0.055)
  MoveL 3353 to (502.78, 490.4, 6.8) mm, rotated rx 0 ry 90 rz 0 deg; joints [-11.076, -26.992, 111.001, -15.077, -83.352, 50.784]
  Call Extruder(0.199)
  MoveL 3354 to (509.6, 490.4, 6.8) mm, rotated rx 0 ry 90 rz 0 deg; joints [-10.955, -26.865, 110.182, -14.977, -82.68, 50.952]
  Call Extruder(0.233)
  MoveL 3355 to (509.6, 498.4, 6.8) mm, rotated rx 0 ry 90 rz 0 deg; joints [-11.679, -26.834, 109.99, -15.713, -82.546, 51.078]
  Call Extruder(0.056)
  MoveL 3356 to (507.66, 498.4, 6.8) mm, rotated rx 0 ry 90 rz 0 deg; joints [-11.716, -26.872, 110.223, -15.743, -82.736, 51.028]
  Set speed (120.0 mm/s)
  MoveL 3357 to (507.66, 498.8, 6.8) mm, rotated rx 0 ry 90 rz 0 deg; joints [-11.752, -26.87, 110.213, -15.779, -82.729, 51.035]
  Set speed (1000.0 mm/s)
  MoveL 3358 to (507.56, 498.8, 6.8) mm, rotated rx 0 ry 90 rz 0 deg; joints [-11.754, -26.872, 110.225, -15.781, -82.739, 51.032]
  Set speed (1000.0 mm/s)
  MoveL 3359 to (499.93, 492.49, 6.8) mm, rotated rx 0 ry 90 rz 0 deg; joints [-11.32, -27.036, 111.291, -15.315, -83.596, 50.743]
  Set speed (15.0 mm/s)
  Call Extruder(0.004)
  MoveL 3360 to (499.74, 492.68, 6.8) mm, rotated rx 0 ry 90 rz 0 deg; joints [-11.341, -27.038, 111.309, -15.336, -83.612, 50.741]
  Set speed (120.0 mm/s)
  MoveL 3361 to (499.25, 492.68, 6.8) mm, rotated rx 0 ry 90 rz 0 deg; joints [-11.35, -27.047, 111.368, -15.343, -83.66, 50.728]
  Set speed (15.0 mm/s)
  Call Extruder(0.014)
  MoveL 3362 to (499.93, 492, 6.8) mm, rotated rx 0 ry 90 rz 0 deg; joints [-11.274, -27.037, 111.303, -15.269, -83.605, 50.736]
  Set speed (120.0 mm/s)
  MoveL 3363 to (499.93, 491.5, 6.8) mm, rotated rx 0 ry 90 rz 0 deg; joints [-11.229, -27.039, 111.315, -15.223, -83.613, 50.729]
  Set speed (15.0 mm/s)
  Call Extruder(0.015)
  MoveL 3364 to (499.2, 492.23, 6.8) mm, rotated rx 0 ry 90 rz 0 deg; joints [-11.31, -27.049, 111.385, -15.303, -83.673, 50.721]
  Set speed (120.0 mm/s)
  MoveL 3365 to (499.2, 491.74, 6.8) mm, rotated rx 0 ry 90 rz 0 deg; joints [-11.264, -27.051, 111.397, -15.256, -83.681, 50.714]
  Set speed (15.0 mm/s)
  MoveL 3366 to (499.93, 491.01, 6.8) mm, rotated rx 0 ry 90 rz 0 deg; joints [-11.183, -27.041, 111.327, -15.177, -83.622, 50.722]
  Set speed (120.0 mm/s)
  MoveL 3367 to (499.71, 490.73, 6.8) mm, rotated rx 0 ry 90 rz 0 deg; joints [-11.162, -27.046, 111.359, -15.154, -83.648, 50.712]
  Set speed (15.0 mm/s)
  Call Extruder(0.011)
  MoveL 3368 to (499.2, 491.24, 6.8) mm, rotated rx 0 ry 90 rz 0 deg; joints [-11.219, -27.053, 111.408, -15.21, -83.69, 50.707]
  Set speed (120.0 mm/s)
  MoveL 3369 to (499.56, 491.25, 6.8) mm, rotated rx 0 ry 90 rz 0 deg; joints [-11.212, -27.046, 111.365, -15.205, -83.654, 50.716]
  Set speed (1000.0 mm/s)
  MoveL 3370 to (496.32, 492.32, 6.8) mm, rotated rx 0 ry 90 rz 0 deg; joints [-11.372, -27.099, 111.725, -15.356, -83.955, 50.649]
  Set speed (1000.0 mm/s)
  MoveL 3371 to (490.68, 490.68, 6.8) mm, rotated rx 0 ry 90 rz 0 deg; joints [-11.324, -27.197, 112.432, -15.292, -84.541, 50.483]
  Set speed (1000.0 mm/s)
  MoveL 3372 to (490.68, 490.68, 6.9) mm, rotated rx 0 ry 90 rz 0 deg; joints [-11.324, -27.207, 112.437, -15.292, -84.536, 50.485]
  Set speed (30.0 mm/s)
  Call Extruder(0.767)
  MoveL 3373 to (509.32, 509.32, 6.9) mm, rotated rx 0 ry 90 rz 0 deg; joints [-12.669, -26.804, 109.745, -16.718, -82.374, 51.254]
  MoveL 3374 to (509.44, 509.44, 6.9) mm, rotated rx 0 ry 90 rz 0 deg; joints [-12.677, -26.801, 109.727, -16.727, -82.36, 51.26]
  Set speed (120.0 mm/s)
  MoveL 3375 to (508.74, 501.16, 6.9) mm, rotated rx 0 ry 90 rz 0 deg; joints [-11.945, -26.85, 110.029, -15.98, -82.577, 51.102]
  Set speed (30.0 mm/s)
  Call Extruder(0.336)
  MoveL 3376 to (500.58, 509.32, 6.9) mm, rotated rx 0 ry 90 rz 0 deg; joints [-12.847, -26.97, 110.791, -16.866, -83.222, 51.018]
  Set speed (120.0 mm/s)
  MoveL 3377 to (499.42, 509.32, 6.9) mm, rotated rx 0 ry 90 rz 0 deg; joints [-12.872, -26.991, 110.929, -16.886, -83.335, 50.986]
  Set speed (30.0 mm/s)
  Call Extruder(0.360)
  MoveL 3378 to (490.68, 500.58, 6.9) mm, rotated rx 0 ry 90 rz 0 deg; joints [-12.247, -27.174, 112.194, -16.225, -84.355, 50.618]
  Set speed (120.0 mm/s)
  MoveL 3379 to (490.68, 499.42, 6.9) mm, rotated rx 0 ry 90 rz 0 deg; joints [-12.139, -27.178, 112.223, -16.116, -84.377, 50.602]
  Set speed (30.0 mm/s)
  Call Extruder(0.282)
  MoveL 3380 to (497.52, 492.57, 6.9) mm, rotated rx 0 ry 90 rz 0 deg; joints [-11.372, -27.088, 111.581, -15.361, -83.827, 50.685]
  MoveL 3381 to (497.65, 492.45, 6.9) mm, rotated rx 0 ry 90 rz 0 deg; joints [-11.359, -27.086, 111.57, -15.347, -83.817, 50.686]
  Set speed (120.0 mm/s)
  MoveL 3382 to (502.48, 492.58, 6.9) mm, rotated rx 0 ry 90 rz 0 deg; joints [-11.281, -27.001, 110.991, -15.284, -83.34, 50.81]
  Set speed (30.0 mm/s)
  Call Extruder(0.228)
  MoveL 3383 to (508.01, 498.12, 6.9) mm, rotated rx 0 ry 90 rz 0 deg; joints [-11.684, -26.877, 110.193, -15.711, -82.701, 51.034]
  MoveL 3384 to (508.14, 498.24, 6.9) mm, rotated rx 0 ry 90 rz 0 deg; joints [-11.692, -26.874, 110.175, -15.721, -82.687, 51.039]
  Set speed (120.0 mm/s)
  MoveL 3385 to (509.32, 490.68, 6.9) mm, rotated rx 0 ry 90 rz 0 deg; joints [-10.985, -26.88, 110.215, -15.007, -82.698, 50.95]
  Set speed (30.0 mm/s)
  Call Extruder(0.767)
  MoveL 3386 to (490.68, 509.32, 6.9) mm, rotated rx 0 ry 90 rz 0 deg; joints [-13.056, -27.142, 111.963, -17.043, -84.185, 50.744]
  MoveL 3387 to (490.56, 509.44, 6.9) mm, rotated rx 0 ry 90 rz 0 deg; joints [-13.07, -27.144, 111.974, -17.057, -84.194, 50.743]
  Set speed (120.0 mm/s)
  MoveL 3388 to (507.59, 498.32, 6.9) mm, rotated rx 0 ry 90 rz 0 deg; joints [-11.711, -26.884, 110.238, -15.737, -82.739, 51.027]
  Set speed (1000.0 mm/s)
  MoveL 3389 to (507.66, 498.4, 6.9) mm, rotated rx 0 ry 90 rz 0 deg; joints [-11.716, -26.882, 110.228, -15.743, -82.731, 51.03]
  Set speed (15.0 mm/s)
  Call Extruder(0.072)
  MoveL 3390 to (507.66, 500.88, 6.9) mm, rotated rx 0 ry 90 rz 0 deg; joints [-11.94, -26.872, 110.166, -15.971, -82.688, 51.07]
  Call Extruder(0.056)
  MoveL 3391 to (509.6, 500.88, 6.9) mm, rotated rx 0 ry 90 rz 0 deg; joints [-11.903, -26.835, 109.933, -15.941, -82.498, 51.12]
  Call Extruder(0.254)
  MoveL 3392 to (509.6, 509.6, 6.9) mm, rotated rx 0 ry 90 rz 0 deg; joints [-12.688, -26.797, 109.704, -16.739, -82.342, 51.266]
  Call Extruder(0.559)
  MoveL 3393 to (490.4, 509.6, 6.9) mm, rotated rx 0 ry 90 rz 0 deg; joints [-13.088, -27.146, 111.988, -17.075, -84.206, 50.741]
  MoveL 3394 to (490.4, 490.4, 6.9) mm, rotated rx 0 ry 90 rz 0 deg; joints [-11.303, -27.213, 112.477, -15.271, -84.568, 50.474]
  Call Extruder(0.175)
  MoveL 3395 to (496.4, 490.4, 6.9) mm, rotated rx 0 ry 90 rz 0 deg; joints [-11.192, -27.114, 111.767, -15.175, -83.975, 50.626]
  Call Extruder(0.055)
  MoveL 3396 to (496.4, 492.3, 6.9) mm, rotated rx 0 ry 90 rz 0 deg; joints [-11.367, -27.108, 111.721, -15.352, -83.942, 50.652]
  Call Extruder(0.063)
  MoveL 3397 to (498.58, 492.29, 6.9) mm, rotated rx 0 ry 90 rz 0 deg; joints [-11.327, -27.07, 111.462, -15.318, -83.728, 50.707]
  Call Extruder(0.010)
  MoveL 3398 to (498.93, 492.29, 6.9) mm, rotated rx 0 ry 90 rz 0 deg; joints [-11.32, -27.064, 111.421, -15.313, -83.693, 50.716]
  Call Extruder(0.007)
  MoveL 3399 to (498.93, 491.94, 6.9) mm, rotated rx 0 ry 90 rz 0 deg; joints [-11.288, -27.066, 111.429, -15.28, -83.699, 50.711]
  Call Extruder(0.035)
  MoveL 3400 to (498.93, 490.75, 6.9) mm, rotated rx 0 ry 90 rz 0 deg; joints [-11.178, -27.07, 111.457, -15.168, -83.72, 50.694]
  Call Extruder(0.010)
  MoveL 3401 to (498.93, 490.4, 6.9) mm, rotated rx 0 ry 90 rz 0 deg; joints [-11.146, -27.071, 111.466, -15.136, -83.726, 50.69]
  Call Extruder(0.007)
  MoveL 3402 to (499.28, 490.4, 6.9) mm, rotated rx 0 ry 90 rz 0 deg; joints [-11.139, -27.065, 111.424, -15.13, -83.691, 50.698]
  Call Extruder(0.027)
  MoveL 3403 to (500.2, 490.4, 6.9) mm, rotated rx 0 ry 90 rz 0 deg; joints [-11.123, -27.049, 111.314, -15.116, -83.6, 50.721]
  Call Extruder(0.055)
  MoveL 3404 to (500.2, 492.3, 6.9) mm, rotated rx 0 ry 90 rz 0 deg; joints [-11.297, -27.042, 111.269, -15.293, -83.568, 50.748]
  Call Extruder(0.073)
  MoveL 3405 to (502.71, 492.3, 6.9) mm, rotated rx 0 ry 90 rz 0 deg; joints [-11.251, -26.997, 110.97, -15.254, -83.321, 50.811]
  Call Extruder(0.055)
  MoveL 3406 to (502.71, 490.4, 6.9) mm, rotated rx 0 ry 90 rz 0 deg; joints [-11.077, -27.004, 111.014, -15.078, -83.353, 50.784]
  Call Extruder(0.200)
  MoveL 3407 to (509.6, 490.4, 6.9) mm, rotated rx 0 ry 90 rz 0 deg; joints [-10.955, -26.876, 110.188, -14.977, -82.675, 50.953]
  Call Extruder(0.233)
  MoveL 3408 to (509.6, 498.4, 6.9) mm, rotated rx 0 ry 90 rz 0 deg; joints [-11.679, -26.845, 109.995, -15.713, -82.541, 51.079]
  Call Extruder(0.056)
  MoveL 3409 to (507.66, 498.4, 6.9) mm, rotated rx 0 ry 90 rz 0 deg; joints [-11.716, -26.882, 110.228, -15.743, -82.731, 51.03]
  Set speed (120.0 mm/s)
  MoveL 3410 to (507.66, 498.8, 6.9) mm, rotated rx 0 ry 90 rz 0 deg; joints [-11.752, -26.881, 110.218, -15.779, -82.724, 51.036]
  Set speed (1000.0 mm/s)
  MoveL 3411 to (507.56, 498.8, 6.9) mm, rotated rx 0 ry 90 rz 0 deg; joints [-11.754, -26.883, 110.23, -15.781, -82.734, 51.034]
  Set speed (1000.0 mm/s)
  MoveL 3412 to (499.87, 492.45, 6.9) mm, rotated rx 0 ry 90 rz 0 deg; joints [-11.317, -27.047, 111.305, -15.312, -83.598, 50.742]
  Set speed (15.0 mm/s)
  Call Extruder(0.013)
  MoveL 3413 to (499.26, 491.84, 6.9) mm, rotated rx 0 ry 90 rz 0 deg; joints [-11.272, -27.06, 111.393, -15.265, -83.669, 50.718]
  Set speed (120.0 mm/s)
  MoveL 3414 to (499.26, 492.33, 6.9) mm, rotated rx 0 ry 90 rz 0 deg; joints [-11.318, -27.059, 111.381, -15.311, -83.66, 50.725]
  Set speed (15.0 mm/s)
  Call Extruder(0.007)
  MoveL 3415 to (499.61, 492.68, 6.9) mm, rotated rx 0 ry 90 rz 0 deg; joints [-11.343, -27.051, 111.331, -15.338, -83.62, 50.739]
  Set speed (120.0 mm/s)
  MoveL 3416 to (499.56, 491.65, 6.9) mm, rotated rx 0 ry 90 rz 0 deg; joints [-11.249, -27.056, 111.361, -15.242, -83.642, 50.723]
  Set speed (15.0 mm/s)
  Call Extruder(0.020)
  MoveL 3417 to (499.57, 491.15, 6.9) mm, rotated rx 0 ry 90 rz 0 deg; joints [-11.203, -27.057, 111.372, -15.196, -83.65, 50.716]
  Call Extruder(0.014)
  MoveL 3418 to (499.75, 490.85, 6.9) mm, rotated rx 0 ry 90 rz 0 deg; joints [-11.172, -27.055, 111.357, -15.165, -83.637, 50.716]
  Set speed (120.0 mm/s)
  MoveL 3419 to (499.5, 491.1, 6.9) mm, rotated rx 0 ry 90 rz 0 deg; joints [-11.2, -27.059, 111.381, -15.192, -83.657, 50.714]
  Set speed (1000.0 mm/s)
  MoveL 3420 to (496.37, 492.32, 6.9) mm, rotated rx 0 ry 90 rz 0 deg; joints [-11.371, -27.108, 111.724, -15.356, -83.945, 50.652]
  Set speed (1000.0 mm/s)
  MoveL 3421 to (490.68, 490.68, 6.9) mm, rotated rx 0 ry 90 rz 0 deg; joints [-11.324, -27.207, 112.437, -15.292, -84.536, 50.485]
  Set speed (1000.0 mm/s)
  MoveL 3422 to (490.68, 490.68, 7) mm, rotated rx 0 ry 90 rz 0 deg; joints [-11.324, -27.218, 112.443, -15.292, -84.531, 50.486]
  Set speed (30.0 mm/s)
  Call Extruder(0.767)
  MoveL 3423 to (509.32, 509.32, 7) mm, rotated rx 0 ry 90 rz 0 deg; joints [-12.669, -26.815, 109.75, -16.718, -82.369, 51.256]
  MoveL 3424 to (509.44, 509.44, 7) mm, rotated rx 0 ry 90 rz 0 deg; joints [-12.677, -26.812, 109.732, -16.727, -82.355, 51.261]
  Set speed (120.0 mm/s)
  MoveL 3425 to (508.74, 501.15, 7) mm, rotated rx 0 ry 90 rz 0 deg; joints [-11.945, -26.861, 110.034, -15.98, -82.572, 51.104]
  Set speed (30.0 mm/s)
  Call Extruder(0.336)
  MoveL 3426 to (500.58, 509.32, 7) mm, rotated rx 0 ry 90 rz 0 deg; joints [-12.847, -26.981, 110.796, -16.866, -83.217, 51.019]
  Set speed (120.0 mm/s)
  MoveL 3427 to (499.42, 509.32, 7) mm, rotated rx 0 ry 90 rz 0 deg; joints [-12.872, -27.002, 110.934, -16.886, -83.33, 50.988]
  Set speed (30.0 mm/s)
  Call Extruder(0.360)
  MoveL 3428 to (490.68, 500.58, 7) mm, rotated rx 0 ry 90 rz 0 deg; joints [-12.247, -27.185, 112.199, -16.225, -84.35, 50.62]
  Set speed (120.0 mm/s)
  MoveL 3429 to (490.68, 499.42, 7) mm, rotated rx 0 ry 90 rz 0 deg; joints [-12.139, -27.189, 112.229, -16.116, -84.371, 50.603]
  Set speed (30.0 mm/s)
  Call Extruder(0.282)
  MoveL 3430 to (497.53, 492.57, 7) mm, rotated rx 0 ry 90 rz 0 deg; joints [-11.372, -27.098, 111.587, -15.361, -83.822, 50.686]
  MoveL 3431 to (497.65, 492.45, 7) mm, rotated rx 0 ry 90 rz 0 deg; joints [-11.359, -27.097, 111.575, -15.348, -83.812, 50.688]
  Set speed (120.0 mm/s)
  MoveL 3432 to (502.47, 492.57, 7) mm, rotated rx 0 ry 90 rz 0 deg; joints [-11.281, -27.011, 110.997, -15.284, -83.335, 50.811]
  Set speed (30.0 mm/s)
  Call Extruder(0.228)
  MoveL 3433 to (508.01, 498.11, 7) mm, rotated rx 0 ry 90 rz 0 deg; joints [-11.683, -26.887, 110.198, -15.711, -82.696, 51.036]
  MoveL 3434 to (508.14, 498.24, 7) mm, rotated rx 0 ry 90 rz 0 deg; joints [-11.692, -26.884, 110.18, -15.721, -82.682, 51.041]
  Set speed (120.0 mm/s)
  MoveL 3435 to (509.32, 490.68, 7) mm, rotated rx 0 ry 90 rz 0 deg; joints [-10.985, -26.891, 110.22, -15.007, -82.693, 50.952]
  Set speed (30.0 mm/s)
  Call Extruder(0.767)
  MoveL 3436 to (490.68, 509.32, 7) mm, rotated rx 0 ry 90 rz 0 deg; joints [-13.056, -27.153, 111.968, -17.044, -84.179, 50.746]
  MoveL 3437 to (490.56, 509.44, 7) mm, rotated rx 0 ry 90 rz 0 deg; joints [-13.07, -27.154, 111.979, -17.057, -84.189, 50.744]
  Set speed (120.0 mm/s)
  MoveL 3438 to (507.59, 498.32, 7) mm, rotated rx 0 ry 90 rz 0 deg; joints [-11.711, -26.894, 110.244, -15.737, -82.734, 51.028]
  Set speed (1000.0 mm/s)
  MoveL 3439 to (507.66, 498.39, 7) mm, rotated rx 0 ry 90 rz 0 deg; joints [-11.716, -26.893, 110.233, -15.743, -82.726, 51.031]
  Set speed (15.0 mm/s)
  Call Extruder(0.072)
  MoveL 3440 to (507.66, 500.87, 7) mm, rotated rx 0 ry 90 rz 0 deg; joints [-11.94, -26.883, 110.171, -15.971, -82.683, 51.071]
  Call Extruder(0.056)
  MoveL 3441 to (509.6, 500.88, 7) mm, rotated rx 0 ry 90 rz 0 deg; joints [-11.903, -26.845, 109.938, -15.941, -82.493, 51.121]
  Call Extruder(0.254)
  MoveL 3442 to (509.6, 509.6, 7) mm, rotated rx 0 ry 90 rz 0 deg; joints [-12.688, -26.808, 109.709, -16.739, -82.337, 51.268]
  Call Extruder(0.559)
  MoveL 3443 to (490.4, 509.6, 7) mm, rotated rx 0 ry 90 rz 0 deg; joints [-13.088, -27.156, 111.993, -17.075, -84.201, 50.742]
  MoveL 3444 to (490.4, 490.4, 7) mm, rotated rx 0 ry 90 rz 0 deg; joints [-11.303, -27.223, 112.482, -15.271, -84.563, 50.476]
  Call Extruder(0.176)
  MoveL 3445 to (496.46, 490.4, 7) mm, rotated rx 0 ry 90 rz 0 deg; joints [-11.191, -27.124, 111.765, -15.174, -83.965, 50.629]
  Call Extruder(0.055)
  MoveL 3446 to (496.46, 492.3, 7) mm, rotated rx 0 ry 90 rz 0 deg; joints [-11.366, -27.118, 111.72, -15.352, -83.932, 50.655]
  Call Extruder(0.074)
  MoveL 3447 to (498.99, 492.29, 7) mm, rotated rx 0 ry 90 rz 0 deg; joints [-11.319, -27.074, 111.419, -15.312, -83.682, 50.719]
  Call Extruder(0.055)
  MoveL 3448 to (498.99, 490.4, 7) mm, rotated rx 0 ry 90 rz 0 deg; joints [-11.145, -27.08, 111.464, -15.135, -83.715, 50.692]
  Call Extruder(0.023)
  MoveL 3449 to (499.79, 490.4, 7) mm, rotated rx 0 ry 90 rz 0 deg; joints [-11.13, -27.066, 111.368, -15.123, -83.636, 50.713]
  Call Extruder(0.010)
  MoveL 3450 to (500.14, 490.4, 7) mm, rotated rx 0 ry 90 rz 0 deg; joints [-11.124, -27.06, 111.326, -15.117, -83.601, 50.721]
  Call Extruder(0.007)
  MoveL 3451 to (500.14, 490.75, 7) mm, rotated rx 0 ry 90 rz 0 deg; joints [-11.156, -27.059, 111.318, -15.15, -83.595, 50.726]
  Call Extruder(0.035)
  MoveL 3452 to (500.14, 491.94, 7) mm, rotated rx 0 ry 90 rz 0 deg; joints [-11.266, -27.055, 111.29, -15.261, -83.575, 50.743]
  Call Extruder(0.010)
  MoveL 3453 to (500.14, 492.3, 7) mm, rotated rx 0 ry 90 rz 0 deg; joints [-11.298, -27.054, 111.282, -15.294, -83.569, 50.748]
  Call Extruder(0.007)
  MoveL 3454 to (500.49, 492.3, 7) mm, rotated rx 0 ry 90 rz 0 deg; joints [-11.292, -27.048, 111.24, -15.289, -83.534, 50.757]
  Call Extruder(0.063)
  MoveL 3455 to (502.65, 492.3, 7) mm, rotated rx 0 ry 90 rz 0 deg; joints [-11.252, -27.009, 110.983, -15.256, -83.322, 50.811]
  Call Extruder(0.055)
  MoveL 3456 to (502.65, 490.4, 7) mm, rotated rx 0 ry 90 rz 0 deg; joints [-11.078, -27.016, 111.027, -15.079, -83.354, 50.783]
  Call Extruder(0.202)
  MoveL 3457 to (509.6, 490.4, 7) mm, rotated rx 0 ry 90 rz 0 deg; joints [-10.955, -26.886, 110.193, -14.977, -82.67, 50.954]
  Call Extruder(0.233)
  MoveL 3458 to (509.6, 498.39, 7) mm, rotated rx 0 ry 90 rz 0 deg; joints [-11.679, -26.855, 110, -15.713, -82.536, 51.081]
  Call Extruder(0.056)
  MoveL 3459 to (507.66, 498.39, 7) mm, rotated rx 0 ry 90 rz 0 deg; joints [-11.716, -26.893, 110.233, -15.743, -82.726, 51.031]
  Set speed (120.0 mm/s)
  MoveL 3460 to (507.66, 498.79, 7) mm, rotated rx 0 ry 90 rz 0 deg; joints [-11.752, -26.891, 110.223, -15.78, -82.719, 51.038]
  Set speed (1000.0 mm/s)
  MoveL 3461 to (507.56, 498.79, 7) mm, rotated rx 0 ry 90 rz 0 deg; joints [-11.754, -26.893, 110.235, -15.781, -82.729, 51.035]
  Set speed (1000.0 mm/s)
  MoveL 3462 to (499.81, 492.61, 7) mm, rotated rx 0 ry 90 rz 0 deg; joints [-11.334, -27.058, 111.314, -15.329, -83.596, 50.744]
  Set speed (1000.0 mm/s)
  MoveL 3463 to (499.78, 492.65, 7) mm, rotated rx 0 ry 90 rz 0 deg; joints [-11.337, -27.059, 111.317, -15.332, -83.599, 50.744]
  Set speed (15.0 mm/s)
  Call Extruder(0.008)
  MoveL 3464 to (499.56, 492.36, 7) mm, rotated rx 0 ry 90 rz 0 deg; joints [-11.315, -27.064, 111.349, -15.309, -83.625, 50.735]
  Call Extruder(0.032)
  MoveL 3465 to (499.52, 490.93, 7) mm, rotated rx 0 ry 90 rz 0 deg; joints [-11.184, -27.069, 111.389, -15.176, -83.654, 50.713]
  Set speed (120.0 mm/s)
  MoveL 3466 to (499.44, 491.12, 7) mm, rotated rx 0 ry 90 rz 0 deg; joints [-11.203, -27.07, 111.393, -15.196, -83.658, 50.714]
  Set speed (1000.0 mm/s)
  MoveL 3467 to (496.43, 492.32, 7) mm, rotated rx 0 ry 90 rz 0 deg; joints [-11.37, -27.118, 111.723, -15.355, -83.934, 50.655]
  Set speed (1000.0 mm/s)
  MoveL 3468 to (490.68, 490.68, 7) mm, rotated rx 0 ry 90 rz 0 deg; joints [-11.324, -27.218, 112.443, -15.292, -84.531, 50.486]
  Set speed (1000.0 mm/s)
  MoveL 3469 to (490.68, 490.68, 7.1) mm, rotated rx 0 ry 90 rz 0 deg; joints [-11.324, -27.229, 112.448, -15.293, -84.526, 50.488]
  Set speed (30.0 mm/s)
  Call Extruder(0.767)
  MoveL 3470 to (509.32, 509.32, 7.1) mm, rotated rx 0 ry 90 rz 0 deg; joints [-12.669, -26.825, 109.756, -16.718, -82.364, 51.257]
  MoveL 3471 to (509.44, 509.44, 7.1) mm, rotated rx 0 ry 90 rz 0 deg; joints [-12.677, -26.822, 109.738, -16.727, -82.35, 51.263]
  Set speed (120.0 mm/s)
  MoveL 3472 to (508.74, 501.15, 7.1) mm, rotated rx 0 ry 90 rz 0 deg; joints [-11.945, -26.871, 110.039, -15.98, -82.567, 51.105]
  Set speed (30.0 mm/s)
  Call Extruder(0.336)
  MoveL 3473 to (500.58, 509.32, 7.1) mm, rotated rx 0 ry 90 rz 0 deg; joints [-12.847, -26.991, 110.801, -16.866, -83.212, 51.021]
  Set speed (120.0 mm/s)
  MoveL 3474 to (499.42, 509.32, 7.1) mm, rotated rx 0 ry 90 rz 0 deg; joints [-12.872, -27.012, 110.939, -16.886, -83.325, 50.989]
  Set speed (30.0 mm/s)
  Call Extruder(0.360)
  MoveL 3475 to (490.68, 500.58, 7.1) mm, rotated rx 0 ry 90 rz 0 deg; joints [-12.247, -27.195, 112.204, -16.225, -84.344, 50.621]
  Set speed (120.0 mm/s)
  MoveL 3476 to (490.68, 499.42, 7.1) mm, rotated rx 0 ry 90 rz 0 deg; joints [-12.139, -27.2, 112.234, -16.116, -84.366, 50.605]
  Set speed (30.0 mm/s)
  Call Extruder(0.282)
  MoveL 3477 to (497.53, 492.57, 7.1) mm, rotated rx 0 ry 90 rz 0 deg; joints [-11.372, -27.109, 111.592, -15.361, -83.817, 50.688]
  MoveL 3478 to (497.65, 492.45, 7.1) mm, rotated rx 0 ry 90 rz 0 deg; joints [-11.359, -27.107, 111.58, -15.348, -83.807, 50.689]
  Set speed (120.0 mm/s)
  MoveL 3479 to (502.47, 492.57, 7.1) mm, rotated rx 0 ry 90 rz 0 deg; joints [-11.281, -27.022, 111.002, -15.284, -83.329, 50.812]
  Set speed (30.0 mm/s)
  Call Extruder(0.228)
  MoveL 3480 to (508.01, 498.11, 7.1) mm, rotated rx 0 ry 90 rz 0 deg; joints [-11.683, -26.898, 110.203, -15.711, -82.691, 51.037]
  MoveL 3481 to (508.13, 498.24, 7.1) mm, rotated rx 0 ry 90 rz 0 deg; joints [-11.692, -26.895, 110.186, -15.721, -82.677, 51.042]
  Set speed (120.0 mm/s)
  MoveL 3482 to (509.32, 490.68, 7.1) mm, rotated rx 0 ry 90 rz 0 deg; joints [-10.985, -26.901, 110.225, -15.007, -82.688, 50.953]
  Set speed (30.0 mm/s)
  Call Extruder(0.767)
  MoveL 3483 to (490.68, 509.32, 7.1) mm, rotated rx 0 ry 90 rz 0 deg; joints [-13.056, -27.163, 111.973, -17.044, -84.174, 50.748]
  MoveL 3484 to (490.56, 509.44, 7.1) mm, rotated rx 0 ry 90 rz 0 deg; joints [-13.07, -27.165, 111.984, -17.058, -84.184, 50.746]
  Set speed (120.0 mm/s)
  MoveL 3485 to (507.59, 498.32, 7.1) mm, rotated rx 0 ry 90 rz 0 deg; joints [-11.71, -26.905, 110.249, -15.737, -82.729, 51.03]
  Set speed (1000.0 mm/s)
  MoveL 3486 to (507.66, 498.39, 7.1) mm, rotated rx 0 ry 90 rz 0 deg; joints [-11.715, -26.903, 110.239, -15.743, -82.721, 51.033]
  Set speed (15.0 mm/s)
  Call Extruder(0.072)
  MoveL 3487 to (507.66, 500.87, 7.1) mm, rotated rx 0 ry 90 rz 0 deg; joints [-11.94, -26.893, 110.176, -15.971, -82.678, 51.072]
  Call Extruder(0.056)
  MoveL 3488 to (509.6, 500.87, 7.1) mm, rotated rx 0 ry 90 rz 0 deg; joints [-11.903, -26.856, 109.943, -15.941, -82.488, 51.122]
  Call Extruder(0.254)
  MoveL 3489 to (509.6, 509.6, 7.1) mm, rotated rx 0 ry 90 rz 0 deg; joints [-12.688, -26.818, 109.714, -16.739, -82.332, 51.27]
  Call Extruder(0.559)
  MoveL 3490 to (490.4, 509.6, 7.1) mm, rotated rx 0 ry 90 rz 0 deg; joints [-13.088, -27.167, 111.998, -17.075, -84.196, 50.744]
  MoveL 3491 to (490.4, 490.4, 7.1) mm, rotated rx 0 ry 90 rz 0 deg; joints [-11.303, -27.234, 112.487, -15.271, -84.558, 50.477]
  Call Extruder(0.178)
  MoveL 3492 to (496.51, 490.4, 7.1) mm, rotated rx 0 ry 90 rz 0 deg; joints [-11.19, -27.134, 111.764, -15.174, -83.954, 50.632]
  Call Extruder(0.055)
  MoveL 3493 to (496.51, 492.3, 7.1) mm, rotated rx 0 ry 90 rz 0 deg; joints [-11.365, -27.127, 111.719, -15.351, -83.921, 50.658]
  Call Extruder(0.064)
  MoveL 3494 to (498.7, 492.29, 7.1) mm, rotated rx 0 ry 90 rz 0 deg; joints [-11.325, -27.09, 111.459, -15.317, -83.706, 50.713]
  Call Extruder(0.010)
  MoveL 3495 to (499.05, 492.29, 7.1) mm, rotated rx 0 ry 90 rz 0 deg; joints [-11.318, -27.083, 111.417, -15.311, -83.671, 50.722]
  Call Extruder(0.007)
  MoveL 3496 to (499.05, 491.94, 7.1) mm, rotated rx 0 ry 90 rz 0 deg; joints [-11.286, -27.085, 111.426, -15.278, -83.677, 50.717]
  Call Extruder(0.045)
  MoveL 3497 to (499.05, 490.4, 7.1) mm, rotated rx 0 ry 90 rz 0 deg; joints [-11.144, -27.09, 111.462, -15.134, -83.704, 50.695]
  Call Extruder(0.030)
  MoveL 3498 to (500.08, 490.4, 7.1) mm, rotated rx 0 ry 90 rz 0 deg; joints [-11.125, -27.072, 111.339, -15.118, -83.602, 50.721]
  Call Extruder(0.045)
  MoveL 3499 to (500.08, 491.95, 7.1) mm, rotated rx 0 ry 90 rz 0 deg; joints [-11.267, -27.067, 111.303, -15.263, -83.576, 50.743]
  Call Extruder(0.010)
  MoveL 3500 to (500.08, 492.3, 7.1) mm, rotated rx 0 ry 90 rz 0 deg; joints [-11.299, -27.065, 111.294, -15.295, -83.57, 50.748]
  Call Extruder(0.007)
  MoveL 3501 to (500.43, 492.3, 7.1) mm, rotated rx 0 ry 90 rz 0 deg; joints [-11.293, -27.059, 111.253, -15.29, -83.535, 50.757]
  Call Extruder(0.063)
  MoveL 3502 to (502.58, 492.29, 7.1) mm, rotated rx 0 ry 90 rz 0 deg; joints [-11.254, -27.021, 110.995, -15.257, -83.323, 50.811]
  Call Extruder(0.055)
  MoveL 3503 to (502.59, 490.4, 7.1) mm, rotated rx 0 ry 90 rz 0 deg; joints [-11.08, -27.027, 111.04, -15.081, -83.355, 50.783]
  Call Extruder(0.204)
  MoveL 3504 to (509.6, 490.4, 7.1) mm, rotated rx 0 ry 90 rz 0 deg; joints [-10.955, -26.897, 110.198, -14.978, -82.665, 50.956]
  Call Extruder(0.233)
  MoveL 3505 to (509.6, 498.39, 7.1) mm, rotated rx 0 ry 90 rz 0 deg; joints [-11.679, -26.866, 110.005, -15.713, -82.531, 51.082]
  Call Extruder(0.056)
  MoveL 3506 to (507.66, 498.39, 7.1) mm, rotated rx 0 ry 90 rz 0 deg; joints [-11.715, -26.903, 110.239, -15.743, -82.721, 51.033]
  Set speed (120.0 mm/s)
  MoveL 3507 to (507.66, 498.79, 7.1) mm, rotated rx 0 ry 90 rz 0 deg; joints [-11.752, -26.902, 110.229, -15.78, -82.714, 51.039]
  Set speed (1000.0 mm/s)
  MoveL 3508 to (507.56, 498.79, 7.1) mm, rotated rx 0 ry 90 rz 0 deg; joints [-11.754, -26.904, 110.241, -15.781, -82.724, 51.036]
  Set speed (1000.0 mm/s)
  MoveL 3509 to (499.61, 492.68, 7.1) mm, rotated rx 0 ry 90 rz 0 deg; joints [-11.343, -27.072, 111.342, -15.338, -83.61, 50.742]
  Set speed (1000.0 mm/s)
  MoveL 3510 to (499.49, 492.56, 7.1) mm, rotated rx 0 ry 90 rz 0 deg; joints [-11.335, -27.075, 111.358, -15.329, -83.623, 50.737]
  Set speed (15.0 mm/s)
  Call Extruder(0.007)
  MoveL 3511 to (499.56, 492.14, 7.1) mm, rotated rx 0 ry 90 rz 0 deg; joints [-11.295, -27.075, 111.36, -15.289, -83.623, 50.733]
  Call Extruder(0.024)
  MoveL 3512 to (499.7, 490.79, 7.1) mm, rotated rx 0 ry 90 rz 0 deg; joints [-11.167, -27.077, 111.376, -15.16, -83.634, 50.717]
  Set speed (120.0 mm/s)
  MoveL 3513 to (499.75, 490.84, 7.1) mm, rotated rx 0 ry 90 rz 0 deg; joints [-11.172, -27.076, 111.368, -15.165, -83.627, 50.719]
  Set speed (1000.0 mm/s)
  MoveL 3514 to (499.08, 492.32, 7.1) mm, rotated rx 0 ry 90 rz 0 deg; joints [-11.32, -27.083, 111.413, -15.313, -83.668, 50.723]
  Set speed (1000.0 mm/s)
  MoveL 3515 to (496.49, 492.32, 7.1) mm, rotated rx 0 ry 90 rz 0 deg; joints [-11.369, -27.128, 111.722, -15.354, -83.924, 50.658]
  Set speed (1000.0 mm/s)
  MoveL 3516 to (490.68, 490.68, 7.1) mm, rotated rx 0 ry 90 rz 0 deg; joints [-11.324, -27.229, 112.448, -15.293, -84.526, 50.488]
  Set speed (1000.0 mm/s)
  MoveL 3517 to (490.68, 490.68, 7.2) mm, rotated rx 0 ry 90 rz 0 deg; joints [-11.324, -27.239, 112.453, -15.293, -84.52, 50.489]
  Set speed (30.0 mm/s)
  Call Extruder(0.767)
  MoveL 3518 to (509.32, 509.32, 7.2) mm, rotated rx 0 ry 90 rz 0 deg; joints [-12.669, -26.836, 109.761, -16.718, -82.359, 51.259]
  MoveL 3519 to (509.44, 509.44, 7.2) mm, rotated rx 0 ry 90 rz 0 deg; joints [-12.677, -26.833, 109.743, -16.728, -82.345, 51.264]
  Set speed (120.0 mm/s)
  MoveL 3520 to (508.74, 501.15, 7.2) mm, rotated rx 0 ry 90 rz 0 deg; joints [-11.945, -26.882, 110.044, -15.98, -82.562, 51.106]
  Set speed (30.0 mm/s)
  Call Extruder(0.336)
  MoveL 3521 to (500.58, 509.32, 7.2) mm, rotated rx 0 ry 90 rz 0 deg; joints [-12.847, -27.002, 110.806, -16.866, -83.207, 51.022]
  Set speed (120.0 mm/s)
  MoveL 3522 to (499.42, 509.32, 7.2) mm, rotated rx 0 ry 90 rz 0 deg; joints [-12.872, -27.023, 110.944, -16.887, -83.32, 50.991]
  Set speed (30.0 mm/s)
  Call Extruder(0.360)
  MoveL 3523 to (490.68, 500.58, 7.2) mm, rotated rx 0 ry 90 rz 0 deg; joints [-12.247, -27.206, 112.21, -16.225, -84.339, 50.623]
  Set speed (120.0 mm/s)
  MoveL 3524 to (490.68, 499.42, 7.2) mm, rotated rx 0 ry 90 rz 0 deg; joints [-12.139, -27.21, 112.239, -16.116, -84.361, 50.606]
  Set speed (30.0 mm/s)
  Call Extruder(0.282)
  MoveL 3525 to (497.52, 492.57, 7.2) mm, rotated rx 0 ry 90 rz 0 deg; joints [-11.372, -27.12, 111.597, -15.361, -83.812, 50.689]
  MoveL 3526 to (497.65, 492.45, 7.2) mm, rotated rx 0 ry 90 rz 0 deg; joints [-11.359, -27.118, 111.586, -15.348, -83.802, 50.69]
  Set speed (120.0 mm/s)
  MoveL 3527 to (502.47, 492.57, 7.2) mm, rotated rx 0 ry 90 rz 0 deg; joints [-11.281, -27.032, 111.007, -15.284, -83.324, 50.814]
  Set speed (30.0 mm/s)
  Call Extruder(0.228)
  MoveL 3528 to (508.01, 498.11, 7.2) mm, rotated rx 0 ry 90 rz 0 deg; joints [-11.683, -26.908, 110.209, -15.712, -82.687, 51.038]
  MoveL 3529 to (508.13, 498.23, 7.2) mm, rotated rx 0 ry 90 rz 0 deg; joints [-11.692, -26.905, 110.191, -15.721, -82.672, 51.044]
  Set speed (120.0 mm/s)
  MoveL 3530 to (509.32, 490.68, 7.2) mm, rotated rx 0 ry 90 rz 0 deg; joints [-10.985, -26.912, 110.231, -15.007, -82.683, 50.955]
  Set speed (30.0 mm/s)
  Call Extruder(0.767)
  MoveL 3531 to (490.68, 509.32, 7.2) mm, rotated rx 0 ry 90 rz 0 deg; joints [-13.056, -27.174, 111.978, -17.044, -84.169, 50.749]
  MoveL 3532 to (490.56, 509.44, 7.2) mm, rotated rx 0 ry 90 rz 0 deg; joints [-13.07, -27.175, 111.99, -17.058, -84.179, 50.747]
  Set speed (120.0 mm/s)
  MoveL 3533 to (507.59, 498.32, 7.2) mm, rotated rx 0 ry 90 rz 0 deg; joints [-11.71, -26.915, 110.254, -15.737, -82.724, 51.031]
  Set speed (1000.0 mm/s)
  MoveL 3534 to (507.66, 498.39, 7.2) mm, rotated rx 0 ry 90 rz 0 deg; joints [-11.715, -26.914, 110.244, -15.743, -82.716, 51.034]
  Set speed (15.0 mm/s)
  Call Extruder(0.072)
  MoveL 3535 to (507.66, 500.87, 7.2) mm, rotated rx 0 ry 90 rz 0 deg; joints [-11.94, -26.904, 110.182, -15.971, -82.673, 51.074]
  Call Extruder(0.056)
  MoveL 3536 to (509.6, 500.87, 7.2) mm, rotated rx 0 ry 90 rz 0 deg; joints [-11.903, -26.866, 109.948, -15.941, -82.483, 51.124]
  Call Extruder(0.254)
  MoveL 3537 to (509.6, 509.6, 7.2) mm, rotated rx 0 ry 90 rz 0 deg; joints [-12.688, -26.829, 109.72, -16.74, -82.327, 51.271]
  Call Extruder(0.559)
  MoveL 3538 to (490.4, 509.6, 7.2) mm, rotated rx 0 ry 90 rz 0 deg; joints [-13.088, -27.177, 112.004, -17.075, -84.191, 50.745]
  MoveL 3539 to (490.4, 490.4, 7.2) mm, rotated rx 0 ry 90 rz 0 deg; joints [-11.303, -27.245, 112.493, -15.271, -84.553, 50.478]
  Call Extruder(0.179)
  MoveL 3540 to (496.57, 490.4, 7.2) mm, rotated rx 0 ry 90 rz 0 deg; joints [-11.189, -27.143, 111.763, -15.173, -83.944, 50.635]
  Call Extruder(0.055)
  MoveL 3541 to (496.57, 492.3, 7.2) mm, rotated rx 0 ry 90 rz 0 deg; joints [-11.364, -27.137, 111.718, -15.35, -83.911, 50.661]
  Call Extruder(0.064)
  MoveL 3542 to (498.76, 492.29, 7.2) mm, rotated rx 0 ry 90 rz 0 deg; joints [-11.324, -27.099, 111.457, -15.316, -83.695, 50.716]
  Call Extruder(0.010)
  MoveL 3543 to (499.11, 492.29, 7.2) mm, rotated rx 0 ry 90 rz 0 deg; joints [-11.317, -27.093, 111.415, -15.31, -83.66, 50.725]
  Call Extruder(0.007)
  MoveL 3544 to (499.11, 491.94, 7.2) mm, rotated rx 0 ry 90 rz 0 deg; joints [-11.285, -27.094, 111.424, -15.278, -83.666, 50.72]
  Call Extruder(0.045)
  MoveL 3545 to (499.11, 490.4, 7.2) mm, rotated rx 0 ry 90 rz 0 deg; joints [-11.142, -27.1, 111.46, -15.133, -83.693, 50.698]
  Call Extruder(0.027)
  MoveL 3546 to (500.02, 490.4, 7.2) mm, rotated rx 0 ry 90 rz 0 deg; joints [-11.126, -27.084, 111.352, -15.12, -83.603, 50.721]
  Call Extruder(0.045)
  MoveL 3547 to (500.02, 491.94, 7.2) mm, rotated rx 0 ry 90 rz 0 deg; joints [-11.268, -27.078, 111.315, -15.264, -83.577, 50.743]
  Call Extruder(0.010)
  MoveL 3548 to (500.02, 492.3, 7.2) mm, rotated rx 0 ry 90 rz 0 deg; joints [-11.301, -27.077, 111.307, -15.296, -83.571, 50.748]
  Call Extruder(0.007)
  MoveL 3549 to (500.37, 492.3, 7.2) mm, rotated rx 0 ry 90 rz 0 deg; joints [-11.294, -27.071, 111.265, -15.291, -83.536, 50.757]
  Call Extruder(0.063)
  MoveL 3550 to (502.52, 492.3, 7.2) mm, rotated rx 0 ry 90 rz 0 deg; joints [-11.255, -27.032, 111.008, -15.258, -83.324, 50.811]
  Call Extruder(0.055)
  MoveL 3551 to (502.52, 490.4, 7.2) mm, rotated rx 0 ry 90 rz 0 deg; joints [-11.081, -27.039, 111.053, -15.082, -83.356, 50.783]
  Call Extruder(0.206)
  MoveL 3552 to (509.6, 490.4, 7.2) mm, rotated rx 0 ry 90 rz 0 deg; joints [-10.955, -26.907, 110.203, -14.978, -82.66, 50.957]
  Call Extruder(0.233)
  MoveL 3553 to (509.6, 498.39, 7.2) mm, rotated rx 0 ry 90 rz 0 deg; joints [-11.679, -26.876, 110.011, -15.713, -82.526, 51.083]
  Call Extruder(0.056)
  MoveL 3554 to (507.66, 498.39, 7.2) mm, rotated rx 0 ry 90 rz 0 deg; joints [-11.715, -26.914, 110.244, -15.743, -82.716, 51.034]
  Set speed (120.0 mm/s)
  MoveL 3555 to (507.66, 498.79, 7.2) mm, rotated rx 0 ry 90 rz 0 deg; joints [-11.752, -26.912, 110.234, -15.78, -82.709, 51.04]
  Set speed (1000.0 mm/s)
  MoveL 3556 to (507.56, 498.79, 7.2) mm, rotated rx 0 ry 90 rz 0 deg; joints [-11.753, -26.914, 110.246, -15.781, -82.719, 51.038]
  Set speed (1000.0 mm/s)
  MoveL 3557 to (499.69, 492.24, 7.2) mm, rotated rx 0 ry 90 rz 0 deg; joints [-11.302, -27.083, 111.348, -15.296, -83.604, 50.739]
  Set speed (1000.0 mm/s)
  MoveL 3558 to (499.56, 492.37, 7.2) mm, rotated rx 0 ry 90 rz 0 deg; joints [-11.315, -27.085, 111.36, -15.31, -83.614, 50.737]
  Set speed (15.0 mm/s)
  Call Extruder(0.007)
  MoveL 3559 to (499.56, 491.87, 7.2) mm, rotated rx 0 ry 90 rz 0 deg; joints [-11.27, -27.087, 111.371, -15.264, -83.623, 50.73]
  Call Extruder(0.013)
  MoveL 3560 to (499.56, 490.88, 7.2) mm, rotated rx 0 ry 90 rz 0 deg; joints [-11.178, -27.09, 111.395, -15.171, -83.64, 50.716]
  Set speed (120.0 mm/s)
  MoveL 3561 to (499.81, 490.76, 7.2) mm, rotated rx 0 ry 90 rz 0 deg; joints [-11.162, -27.086, 111.368, -15.156, -83.618, 50.721]
  Set speed (1000.0 mm/s)
  MoveL 3562 to (499.14, 492.32, 7.2) mm, rotated rx 0 ry 90 rz 0 deg; joints [-11.319, -27.092, 111.411, -15.312, -83.657, 50.726]
  Set speed (1000.0 mm/s)
  MoveL 3563 to (496.54, 492.32, 7.2) mm, rotated rx 0 ry 90 rz 0 deg; joints [-11.367, -27.137, 111.72, -15.353, -83.913, 50.66]
  Set speed (1000.0 mm/s)
  MoveL 3564 to (490.68, 490.68, 7.2) mm, rotated rx 0 ry 90 rz 0 deg; joints [-11.324, -27.239, 112.453, -15.293, -84.52, 50.489]
  Set speed (1000.0 mm/s)
  MoveL 3565 to (490.68, 490.68, 7.3) mm, rotated rx 0 ry 90 rz 0 deg; joints [-11.324, -27.25, 112.459, -15.293, -84.515, 50.491]
  Set speed (30.0 mm/s)
  Call Extruder(0.767)
  MoveL 3566 to (509.32, 509.32, 7.3) mm, rotated rx 0 ry 90 rz 0 deg; joints [-12.669, -26.846, 109.766, -16.719, -82.354, 51.26]
  MoveL 3567 to (509.44, 509.44, 7.3) mm, rotated rx 0 ry 90 rz 0 deg; joints [-12.677, -26.843, 109.748, -16.728, -82.34, 51.266]
  Set speed (120.0 mm/s)
  MoveL 3568 to (508.75, 501.15, 7.3) mm, rotated rx 0 ry 90 rz 0 deg; joints [-11.944, -26.892, 110.049, -15.98, -82.557, 51.108]
  Set speed (30.0 mm/s)
  Call Extruder(0.336)
  MoveL 3569 to (500.58, 509.32, 7.3) mm, rotated rx 0 ry 90 rz 0 deg; joints [-12.847, -27.012, 110.812, -16.867, -83.202, 51.024]
  Set speed (120.0 mm/s)
  MoveL 3570 to (499.42, 509.32, 7.3) mm, rotated rx 0 ry 90 rz 0 deg; joints [-12.872, -27.033, 110.95, -16.887, -83.315, 50.992]
  Set speed (30.0 mm/s)
  Call Extruder(0.360)
  MoveL 3571 to (490.68, 500.58, 7.3) mm, rotated rx 0 ry 90 rz 0 deg; joints [-12.247, -27.217, 112.215, -16.225, -84.334, 50.624]
  Set speed (120.0 mm/s)
  MoveL 3572 to (490.68, 499.42, 7.3) mm, rotated rx 0 ry 90 rz 0 deg; joints [-12.139, -27.221, 112.244, -16.116, -84.356, 50.608]
  Set speed (30.0 mm/s)
  Call Extruder(0.282)
  MoveL 3573 to (497.52, 492.57, 7.3) mm, rotated rx 0 ry 90 rz 0 deg; joints [-11.372, -27.13, 111.603, -15.361, -83.807, 50.69]
  MoveL 3574 to (497.65, 492.45, 7.3) mm, rotated rx 0 ry 90 rz 0 deg; joints [-11.359, -27.128, 111.591, -15.348, -83.797, 50.692]
  Set speed (120.0 mm/s)
  MoveL 3575 to (502.47, 492.57, 7.3) mm, rotated rx 0 ry 90 rz 0 deg; joints [-11.281, -27.043, 111.013, -15.285, -83.319, 50.815]
  Set speed (30.0 mm/s)
  Call Extruder(0.228)
  MoveL 3576 to (508.01, 498.11, 7.3) mm, rotated rx 0 ry 90 rz 0 deg; joints [-11.683, -26.919, 110.214, -15.712, -82.682, 51.04]
  MoveL 3577 to (508.13, 498.23, 7.3) mm, rotated rx 0 ry 90 rz 0 deg; joints [-11.692, -26.916, 110.196, -15.721, -82.667, 51.045]
  Set speed (120.0 mm/s)
  MoveL 3578 to (509.32, 490.68, 7.3) mm, rotated rx 0 ry 90 rz 0 deg; joints [-10.985, -26.922, 110.236, -15.008, -82.678, 50.956]
  Set speed (30.0 mm/s)
  Call Extruder(0.767)
  MoveL 3579 to (490.68, 509.32, 7.3) mm, rotated rx 0 ry 90 rz 0 deg; joints [-13.056, -27.185, 111.984, -17.044, -84.164, 50.751]
  MoveL 3580 to (490.56, 509.44, 7.3) mm, rotated rx 0 ry 90 rz 0 deg; joints [-13.07, -27.186, 111.995, -17.058, -84.174, 50.749]
  Set speed (120.0 mm/s)
  MoveL 3581 to (507.59, 498.32, 7.3) mm, rotated rx 0 ry 90 rz 0 deg; joints [-11.71, -26.926, 110.259, -15.738, -82.719, 51.033]
  Set speed (1000.0 mm/s)
  MoveL 3582 to (507.66, 498.39, 7.3) mm, rotated rx 0 ry 90 rz 0 deg; joints [-11.715, -26.924, 110.249, -15.743, -82.711, 51.035]
  Set speed (15.0 mm/s)
  Call Extruder(0.072)
  MoveL 3583 to (507.66, 500.87, 7.3) mm, rotated rx 0 ry 90 rz 0 deg; joints [-11.94, -26.914, 110.187, -15.971, -82.668, 51.075]
  Call Extruder(0.056)
  MoveL 3584 to (509.6, 500.87, 7.3) mm, rotated rx 0 ry 90 rz 0 deg; joints [-11.903, -26.877, 109.954, -15.941, -82.478, 51.125]
  Call Extruder(0.254)
  MoveL 3585 to (509.6, 509.6, 7.3) mm, rotated rx 0 ry 90 rz 0 deg; joints [-12.688, -26.839, 109.725, -16.74, -82.322, 51.273]
  Call Extruder(0.559)
  MoveL 3586 to (490.4, 509.6, 7.3) mm, rotated rx 0 ry 90 rz 0 deg; joints [-13.088, -27.188, 112.009, -17.075, -84.186, 50.747]
  MoveL 3587 to (490.4, 490.4, 7.3) mm, rotated rx 0 ry 90 rz 0 deg; joints [-11.303, -27.255, 112.498, -15.271, -84.548, 50.48]
  Call Extruder(0.181)
  MoveL 3588 to (496.62, 490.4, 7.3) mm, rotated rx 0 ry 90 rz 0 deg; joints [-11.188, -27.153, 111.761, -15.172, -83.933, 50.637]
  Call Extruder(0.055)
  MoveL 3589 to (496.62, 492.3, 7.3) mm, rotated rx 0 ry 90 rz 0 deg; joints [-11.363, -27.147, 111.716, -15.35, -83.9, 50.664]
  Call Extruder(0.064)
  MoveL 3590 to (498.82, 492.29, 7.3) mm, rotated rx 0 ry 90 rz 0 deg; joints [-11.323, -27.109, 111.455, -15.315, -83.684, 50.719]
  Call Extruder(0.010)
  MoveL 3591 to (499.17, 492.29, 7.3) mm, rotated rx 0 ry 90 rz 0 deg; joints [-11.316, -27.103, 111.414, -15.31, -83.649, 50.728]
  Call Extruder(0.007)
  MoveL 3592 to (499.17, 491.94, 7.3) mm, rotated rx 0 ry 90 rz 0 deg; joints [-11.284, -27.104, 111.422, -15.277, -83.655, 50.723]
  Call Extruder(0.045)
  MoveL 3593 to (499.17, 490.4, 7.3) mm, rotated rx 0 ry 90 rz 0 deg; joints [-11.141, -27.109, 111.459, -15.133, -83.682, 50.701]
  Call Extruder(0.023)
  MoveL 3594 to (499.96, 490.4, 7.3) mm, rotated rx 0 ry 90 rz 0 deg; joints [-11.127, -27.095, 111.364, -15.121, -83.604, 50.721]
  Call Extruder(0.045)
  MoveL 3595 to (499.96, 491.95, 7.3) mm, rotated rx 0 ry 90 rz 0 deg; joints [-11.269, -27.09, 111.328, -15.265, -83.578, 50.743]
  Call Extruder(0.010)
  MoveL 3596 to (499.96, 492.3, 7.3) mm, rotated rx 0 ry 90 rz 0 deg; joints [-11.302, -27.089, 111.319, -15.297, -83.572, 50.748]
  Call Extruder(0.007)
  MoveL 3597 to (500.31, 492.3, 7.3) mm, rotated rx 0 ry 90 rz 0 deg; joints [-11.295, -27.082, 111.278, -15.292, -83.537, 50.757]
  Call Extruder(0.063)
  MoveL 3598 to (502.46, 492.3, 7.3) mm, rotated rx 0 ry 90 rz 0 deg; joints [-11.256, -27.044, 111.021, -15.259, -83.326, 50.811]
  Call Extruder(0.055)
  MoveL 3599 to (502.46, 490.4, 7.3) mm, rotated rx 0 ry 90 rz 0 deg; joints [-11.082, -27.051, 111.066, -15.083, -83.357, 50.783]
  Call Extruder(0.208)
  MoveL 3600 to (509.6, 490.4, 7.3) mm, rotated rx 0 ry 90 rz 0 deg; joints [-10.955, -26.918, 110.209, -14.978, -82.654, 50.958]
  Call Extruder(0.233)
  MoveL 3601 to (509.6, 498.39, 7.3) mm, rotated rx 0 ry 90 rz 0 deg; joints [-11.679, -26.887, 110.016, -15.713, -82.521, 51.085]
  Call Extruder(0.056)
  MoveL 3602 to (507.66, 498.39, 7.3) mm, rotated rx 0 ry 90 rz 0 deg; joints [-11.715, -26.924, 110.249, -15.743, -82.711, 51.035]
  Set speed (120.0 mm/s)
  MoveL 3603 to (507.66, 498.79, 7.3) mm, rotated rx 0 ry 90 rz 0 deg; joints [-11.751, -26.923, 110.239, -15.78, -82.704, 51.042]
  Set speed (1000.0 mm/s)
  MoveL 3604 to (507.56, 498.79, 7.3) mm, rotated rx 0 ry 90 rz 0 deg; joints [-11.753, -26.925, 110.251, -15.781, -82.714, 51.039]
  Set speed (1000.0 mm/s)
  MoveL 3605 to (499.61, 492.68, 7.3) mm, rotated rx 0 ry 90 rz 0 deg; joints [-11.343, -27.093, 111.352, -15.339, -83.6, 50.745]
  Set speed (1000.0 mm/s)
  MoveL 3606 to (499.55, 492.62, 7.3) mm, rotated rx 0 ry 90 rz 0 deg; joints [-11.339, -27.095, 111.36, -15.334, -83.606, 50.742]
  Set speed (15.0 mm/s)
  Call Extruder(0.003)
  MoveL 3607 to (499.56, 492.14, 7.3) mm, rotated rx 0 ry 90 rz 0 deg; joints [-11.294, -27.096, 111.37, -15.289, -83.613, 50.736]
  Call Extruder(0.007)
  MoveL 3608 to (499.56, 491.15, 7.3) mm, rotated rx 0 ry 90 rz 0 deg; joints [-11.203, -27.1, 111.394, -15.197, -83.63, 50.722]
  Set speed (120.0 mm/s)
  MoveL 3609 to (499.26, 491.08, 7.3) mm, rotated rx 0 ry 90 rz 0 deg; joints [-11.203, -27.105, 111.431, -15.195, -83.661, 50.713]
  Set speed (1000.0 mm/s)
  MoveL 3610 to (499.27, 491.08, 7.3) mm, rotated rx 0 ry 90 rz 0 deg; joints [-11.203, -27.105, 111.43, -15.195, -83.66, 50.713]
  Set speed (1000.0 mm/s)
  MoveL 3611 to (496.6, 492.32, 7.3) mm, rotated rx 0 ry 90 rz 0 deg; joints [-11.366, -27.147, 111.719, -15.353, -83.902, 50.663]
  Set speed (1000.0 mm/s)
  MoveL 3612 to (490.68, 490.68, 7.3) mm, rotated rx 0 ry 90 rz 0 deg; joints [-11.324, -27.25, 112.459, -15.293, -84.515, 50.491]
  Set speed (1000.0 mm/s)
  MoveL 3613 to (490.68, 490.68, 7.4) mm, rotated rx 0 ry 90 rz 0 deg; joints [-11.324, -27.261, 112.464, -15.293, -84.51, 50.492]
  Set speed (30.0 mm/s)
  Call Extruder(0.767)
  MoveL 3614 to (509.32, 509.32, 7.4) mm, rotated rx 0 ry 90 rz 0 deg; joints [-12.669, -26.856, 109.771, -16.719, -82.349, 51.262]
  MoveL 3615 to (509.44, 509.44, 7.4) mm, rotated rx 0 ry 90 rz 0 deg; joints [-12.677, -26.853, 109.753, -16.728, -82.335, 51.267]
  Set speed (120.0 mm/s)
  MoveL 3616 to (508.75, 501.15, 7.4) mm, rotated rx 0 ry 90 rz 0 deg; joints [-11.944, -26.903, 110.054, -15.98, -82.551, 51.109]
  Set speed (30.0 mm/s)
  Call Extruder(0.336)
  MoveL 3617 to (500.58, 509.32, 7.4) mm, rotated rx 0 ry 90 rz 0 deg; joints [-12.847, -27.023, 110.817, -16.867, -83.197, 51.026]
  Set speed (120.0 mm/s)
  MoveL 3618 to (499.42, 509.32, 7.4) mm, rotated rx 0 ry 90 rz 0 deg; joints [-12.872, -27.044, 110.955, -16.887, -83.309, 50.994]
  Set speed (30.0 mm/s)
  Call Extruder(0.360)
  MoveL 3619 to (490.68, 500.58, 7.4) mm, rotated rx 0 ry 90 rz 0 deg; joints [-12.247, -27.227, 112.22, -16.225, -84.329, 50.626]
  Set speed (120.0 mm/s)
  MoveL 3620 to (490.68, 499.42, 7.4) mm, rotated rx 0 ry 90 rz 0 deg; joints [-12.139, -27.231, 112.25, -16.116, -84.351, 50.609]
  Set speed (30.0 mm/s)
  Call Extruder(0.282)
  MoveL 3621 to (497.53, 492.57, 7.4) mm, rotated rx 0 ry 90 rz 0 deg; joints [-11.372, -27.141, 111.608, -15.362, -83.801, 50.692]
  MoveL 3622 to (497.65, 492.45, 7.4) mm, rotated rx 0 ry 90 rz 0 deg; joints [-11.359, -27.139, 111.596, -15.348, -83.791, 50.693]
  Set speed (120.0 mm/s)
  MoveL 3623 to (502.47, 492.57, 7.4) mm, rotated rx 0 ry 90 rz 0 deg; joints [-11.281, -27.053, 111.018, -15.285, -83.314, 50.817]
  Set speed (30.0 mm/s)
  Call Extruder(0.228)
  MoveL 3624 to (508.01, 498.11, 7.4) mm, rotated rx 0 ry 90 rz 0 deg; joints [-11.683, -26.929, 110.22, -15.712, -82.677, 51.041]
  MoveL 3625 to (508.13, 498.23, 7.4) mm, rotated rx 0 ry 90 rz 0 deg; joints [-11.692, -26.926, 110.202, -15.721, -82.663, 51.046]
  Set speed (120.0 mm/s)
  MoveL 3626 to (509.32, 490.68, 7.4) mm, rotated rx 0 ry 90 rz 0 deg; joints [-10.985, -26.933, 110.241, -15.008, -82.673, 50.957]
  Set speed (30.0 mm/s)
  Call Extruder(0.767)
  MoveL 3627 to (490.68, 509.32, 7.4) mm, rotated rx 0 ry 90 rz 0 deg; joints [-13.056, -27.195, 111.989, -17.044, -84.159, 50.752]
  MoveL 3628 to (490.56, 509.44, 7.4) mm, rotated rx 0 ry 90 rz 0 deg; joints [-13.07, -27.197, 112, -17.058, -84.169, 50.751]
  Set speed (120.0 mm/s)
  MoveL 3629 to (499.83, 492.37, 7.4) mm, rotated rx 0 ry 90 rz 0 deg; joints [-11.31, -27.101, 111.339, -15.306, -83.578, 50.747]
  Set speed (1000.0 mm/s)
  MoveL 3630 to (499.9, 492.29, 7.4) mm, rotated rx 0 ry 90 rz 0 deg; joints [-11.303, -27.1, 111.332, -15.298, -83.572, 50.748]
  Set speed (15.0 mm/s)
  Call Extruder(0.010)
  MoveL 3631 to (500.25, 492.3, 7.4) mm, rotated rx 0 ry 90 rz 0 deg; joints [-11.296, -27.094, 111.29, -15.293, -83.538, 50.757]
  Call Extruder(0.062)
  MoveL 3632 to (502.39, 492.3, 7.4) mm, rotated rx 0 ry 90 rz 0 deg; joints [-11.257, -27.056, 111.034, -15.26, -83.327, 50.81]
  Call Extruder(0.055)
  MoveL 3633 to (502.4, 490.4, 7.4) mm, rotated rx 0 ry 90 rz 0 deg; joints [-11.083, -27.062, 111.078, -15.084, -83.358, 50.783]
  Call Extruder(0.210)
  MoveL 3634 to (509.6, 490.4, 7.4) mm, rotated rx 0 ry 90 rz 0 deg; joints [-10.955, -26.928, 110.214, -14.978, -82.649, 50.96]
  Call Extruder(0.233)
  MoveL 3635 to (509.6, 498.39, 7.4) mm, rotated rx 0 ry 90 rz 0 deg; joints [-11.679, -26.897, 110.021, -15.713, -82.516, 51.086]
  Call Extruder(0.056)
  MoveL 3636 to (507.66, 498.39, 7.4) mm, rotated rx 0 ry 90 rz 0 deg; joints [-11.715, -26.935, 110.255, -15.743, -82.706, 51.037]
  Call Extruder(0.072)
  MoveL 3637 to (507.66, 500.87, 7.4) mm, rotated rx 0 ry 90 rz 0 deg; joints [-11.94, -26.925, 110.192, -15.971, -82.663, 51.077]
  Call Extruder(0.056)
  MoveL 3638 to (509.6, 500.87, 7.4) mm, rotated rx 0 ry 90 rz 0 deg; joints [-11.903, -26.887, 109.959, -15.941, -82.473, 51.127]
  Call Extruder(0.254)
  MoveL 3639 to (509.6, 509.6, 7.4) mm, rotated rx 0 ry 90 rz 0 deg; joints [-12.688, -26.85, 109.73, -16.74, -82.317, 51.274]
  Call Extruder(0.559)
  MoveL 3640 to (490.4, 509.6, 7.4) mm, rotated rx 0 ry 90 rz 0 deg; joints [-13.088, -27.199, 112.014, -17.076, -84.181, 50.749]
  MoveL 3641 to (490.4, 490.4, 7.4) mm, rotated rx 0 ry 90 rz 0 deg; joints [-11.303, -27.266, 112.503, -15.271, -84.543, 50.481]
  Call Extruder(0.183)
  MoveL 3642 to (496.68, 490.4, 7.4) mm, rotated rx 0 ry 90 rz 0 deg; joints [-11.187, -27.163, 111.76, -15.171, -83.922, 50.64]
  Call Extruder(0.055)
  MoveL 3643 to (496.68, 492.3, 7.4) mm, rotated rx 0 ry 90 rz 0 deg; joints [-11.362, -27.156, 111.715, -15.349, -83.89, 50.666]
  Call Extruder(0.074)
  MoveL 3644 to (499.23, 492.29, 7.4) mm, rotated rx 0 ry 90 rz 0 deg; joints [-11.315, -27.112, 111.412, -15.309, -83.639, 50.731]
  Call Extruder(0.025)
  MoveL 3645 to (499.23, 491.42, 7.4) mm, rotated rx 0 ry 90 rz 0 deg; joints [-11.235, -27.115, 111.433, -15.227, -83.653, 50.718]
  Call Extruder(0.030)
  MoveL 3646 to (499.23, 490.4, 7.4) mm, rotated rx 0 ry 90 rz 0 deg; joints [-11.14, -27.119, 111.457, -15.132, -83.671, 50.704]
  Call Extruder(0.020)
  MoveL 3647 to (499.9, 490.4, 7.4) mm, rotated rx 0 ry 90 rz 0 deg; joints [-11.128, -27.107, 111.377, -15.122, -83.605, 50.721]
  Call Extruder(0.029)
  MoveL 3648 to (499.9, 491.42, 7.4) mm, rotated rx 0 ry 90 rz 0 deg; joints [-11.222, -27.103, 111.353, -15.217, -83.587, 50.735]
  Call Extruder(0.015)
  MoveL 3649 to (499.9, 491.95, 7.4) mm, rotated rx 0 ry 90 rz 0 deg; joints [-11.271, -27.102, 111.34, -15.266, -83.578, 50.743]
  Call Extruder(0.007)
  MoveL 3650 to (499.9, 492.29, 7.4) mm, rotated rx 0 ry 90 rz 0 deg; joints [-11.303, -27.1, 111.332, -15.298, -83.572, 50.748]
  Set speed (120.0 mm/s)
  MoveL 3651 to (500.25, 492.3, 7.4) mm, rotated rx 0 ry 90 rz 0 deg; joints [-11.296, -27.094, 111.29, -15.293, -83.538, 50.757]
  Set speed (1000.0 mm/s)
  MoveL 3652 to (500.3, 492.29, 7.4) mm, rotated rx 0 ry 90 rz 0 deg; joints [-11.295, -27.093, 111.284, -15.292, -83.533, 50.758]
  Set speed (1000.0 mm/s)
  MoveL 3653 to (500.3, 493, 7.4) mm, rotated rx 0 ry 90 rz 0 deg; joints [-11.36, -27.091, 111.268, -15.357, -83.521, 50.768]
  Set speed (1000.0 mm/s)
  MoveL 3654 to (497.02, 492.39, 7.4) mm, rotated rx 0 ry 90 rz 0 deg; joints [-11.365, -27.15, 111.673, -15.353, -83.855, 50.676]
  Set speed (1000.0 mm/s)
  MoveL 3655 to (490.68, 490.68, 7.4) mm, rotated rx 0 ry 90 rz 0 deg; joints [-11.324, -27.261, 112.464, -15.293, -84.51, 50.492]
  Set speed (1000.0 mm/s)
  MoveL 3656 to (490.68, 490.68, 7.5) mm, rotated rx 0 ry 90 rz 0 deg; joints [-11.324, -27.271, 112.469, -15.293, -84.505, 50.493]
  Set speed (30.0 mm/s)
  Call Extruder(0.767)
  MoveL 3657 to (509.32, 509.32, 7.5) mm, rotated rx 0 ry 90 rz 0 deg; joints [-12.669, -26.867, 109.777, -16.719, -82.344, 51.263]
  MoveL 3658 to (509.44, 509.44, 7.5) mm, rotated rx 0 ry 90 rz 0 deg; joints [-12.677, -26.864, 109.758, -16.728, -82.33, 51.269]
  Set speed (120.0 mm/s)
  MoveL 3659 to (508.75, 501.15, 7.5) mm, rotated rx 0 ry 90 rz 0 deg; joints [-11.944, -26.913, 110.059, -15.98, -82.546, 51.111]
  Set speed (30.0 mm/s)
  Call Extruder(0.336)
  MoveL 3660 to (500.58, 509.32, 7.5) mm, rotated rx 0 ry 90 rz 0 deg; joints [-12.847, -27.033, 110.822, -16.867, -83.192, 51.027]
  Set speed (120.0 mm/s)
  MoveL 3661 to (499.42, 509.32, 7.5) mm, rotated rx 0 ry 90 rz 0 deg; joints [-12.872, -27.054, 110.96, -16.887, -83.304, 50.995]
  Set speed (30.0 mm/s)
  Call Extruder(0.360)
  MoveL 3662 to (490.68, 500.58, 7.5) mm, rotated rx 0 ry 90 rz 0 deg; joints [-12.247, -27.238, 112.225, -16.226, -84.324, 50.627]
  Set speed (120.0 mm/s)
  MoveL 3663 to (490.68, 499.42, 7.5) mm, rotated rx 0 ry 90 rz 0 deg; joints [-12.139, -27.242, 112.255, -16.117, -84.346, 50.611]
  Set speed (30.0 mm/s)
  Call Extruder(0.282)
  MoveL 3664 to (497.52, 492.57, 7.5) mm, rotated rx 0 ry 90 rz 0 deg; joints [-11.373, -27.151, 111.613, -15.362, -83.796, 50.693]
  MoveL 3665 to (497.65, 492.45, 7.5) mm, rotated rx 0 ry 90 rz 0 deg; joints [-11.359, -27.15, 111.602, -15.348, -83.786, 50.695]
  Set speed (120.0 mm/s)
  MoveL 3666 to (502.48, 492.58, 7.5) mm, rotated rx 0 ry 90 rz 0 deg; joints [-11.281, -27.064, 111.023, -15.285, -83.309, 50.818]
  Set speed (30.0 mm/s)
  Call Extruder(0.228)
  MoveL 3667 to (508.01, 498.11, 7.5) mm, rotated rx 0 ry 90 rz 0 deg; joints [-11.683, -26.94, 110.225, -15.712, -82.672, 51.043]
  MoveL 3668 to (508.13, 498.23, 7.5) mm, rotated rx 0 ry 90 rz 0 deg; joints [-11.692, -26.937, 110.207, -15.721, -82.658, 51.048]
  Set speed (120.0 mm/s)
  MoveL 3669 to (509.32, 490.68, 7.5) mm, rotated rx 0 ry 90 rz 0 deg; joints [-10.985, -26.943, 110.246, -15.008, -82.667, 50.959]
  Set speed (30.0 mm/s)
  Call Extruder(0.767)
  MoveL 3670 to (490.68, 509.32, 7.5) mm, rotated rx 0 ry 90 rz 0 deg; joints [-13.056, -27.206, 111.994, -17.044, -84.154, 50.754]
  MoveL 3671 to (490.56, 509.44, 7.5) mm, rotated rx 0 ry 90 rz 0 deg; joints [-13.07, -27.207, 112.005, -17.058, -84.163, 50.752]
  Set speed (120.0 mm/s)
  MoveL 3672 to (499.77, 492.37, 7.5) mm, rotated rx 0 ry 90 rz 0 deg; joints [-11.312, -27.113, 111.351, -15.307, -83.579, 50.747]
  Set speed (1000.0 mm/s)
  MoveL 3673 to (499.84, 492.3, 7.5) mm, rotated rx 0 ry 90 rz 0 deg; joints [-11.304, -27.112, 111.344, -15.3, -83.573, 50.748]
  Set speed (15.0 mm/s)
  Call Extruder(0.010)
  MoveL 3674 to (500.19, 492.3, 7.5) mm, rotated rx 0 ry 90 rz 0 deg; joints [-11.297, -27.106, 111.303, -15.294, -83.539, 50.756]
  Call Extruder(0.062)
  MoveL 3675 to (502.33, 492.3, 7.5) mm, rotated rx 0 ry 90 rz 0 deg; joints [-11.258, -27.067, 111.047, -15.261, -83.328, 50.81]
  Call Extruder(0.055)
  MoveL 3676 to (502.33, 490.4, 7.5) mm, rotated rx 0 ry 90 rz 0 deg; joints [-11.084, -27.074, 111.091, -15.085, -83.36, 50.783]
  Call Extruder(0.211)
  MoveL 3677 to (509.6, 490.4, 7.5) mm, rotated rx 0 ry 90 rz 0 deg; joints [-10.955, -26.939, 110.219, -14.978, -82.644, 50.961]
  Call Extruder(0.232)
  MoveL 3678 to (509.6, 498.39, 7.5) mm, rotated rx 0 ry 90 rz 0 deg; joints [-11.679, -26.908, 110.026, -15.713, -82.511, 51.088]
  Call Extruder(0.056)
  MoveL 3679 to (507.66, 498.39, 7.5) mm, rotated rx 0 ry 90 rz 0 deg; joints [-11.715, -26.945, 110.26, -15.743, -82.701, 51.038]
  Call Extruder(0.072)
  MoveL 3680 to (507.66, 500.87, 7.5) mm, rotated rx 0 ry 90 rz 0 deg; joints [-11.94, -26.935, 110.197, -15.971, -82.658, 51.078]
  Call Extruder(0.056)
  MoveL 3681 to (509.6, 500.87, 7.5) mm, rotated rx 0 ry 90 rz 0 deg; joints [-11.903, -26.898, 109.964, -15.941, -82.468, 51.128]
  Call Extruder(0.254)
  MoveL 3682 to (509.6, 509.6, 7.5) mm, rotated rx 0 ry 90 rz 0 deg; joints [-12.688, -26.86, 109.735, -16.74, -82.312, 51.276]
  Call Extruder(0.559)
  MoveL 3683 to (490.4, 509.6, 7.5) mm, rotated rx 0 ry 90 rz 0 deg; joints [-13.088, -27.209, 112.019, -17.076, -84.175, 50.75]
  MoveL 3684 to (490.4, 490.4, 7.5) mm, rotated rx 0 ry 90 rz 0 deg; joints [-11.303, -27.277, 112.509, -15.271, -84.537, 50.483]
  Call Extruder(0.184)
  MoveL 3685 to (496.73, 490.4, 7.5) mm, rotated rx 0 ry 90 rz 0 deg; joints [-11.186, -27.172, 111.759, -15.171, -83.912, 50.643]
  Call Extruder(0.055)
  MoveL 3686 to (496.74, 492.3, 7.5) mm, rotated rx 0 ry 90 rz 0 deg; joints [-11.361, -27.166, 111.714, -15.348, -83.879, 50.669]
  Call Extruder(0.074)
  MoveL 3687 to (499.29, 492.29, 7.5) mm, rotated rx 0 ry 90 rz 0 deg; joints [-11.314, -27.122, 111.41, -15.308, -83.628, 50.734]
  Call Extruder(0.024)
  MoveL 3688 to (499.29, 491.46, 7.5) mm, rotated rx 0 ry 90 rz 0 deg; joints [-11.237, -27.125, 111.43, -15.23, -83.642, 50.722]
  Call Extruder(0.031)
  MoveL 3689 to (499.29, 490.4, 7.5) mm, rotated rx 0 ry 90 rz 0 deg; joints [-11.139, -27.128, 111.455, -15.131, -83.66, 50.707]
  Call Extruder(0.016)
  MoveL 3690 to (499.84, 490.4, 7.5) mm, rotated rx 0 ry 90 rz 0 deg; joints [-11.129, -27.119, 111.389, -15.123, -83.605, 50.721]
  Call Extruder(0.024)
  MoveL 3691 to (499.84, 491.46, 7.5) mm, rotated rx 0 ry 90 rz 0 deg; joints [-11.227, -27.115, 111.364, -15.222, -83.588, 50.736]
  Call Extruder(0.014)
  MoveL 3692 to (499.84, 491.95, 7.5) mm, rotated rx 0 ry 90 rz 0 deg; joints [-11.272, -27.113, 111.353, -15.267, -83.579, 50.743]
  Call Extruder(0.007)
  MoveL 3693 to (499.84, 492.3, 7.5) mm, rotated rx 0 ry 90 rz 0 deg; joints [-11.304, -27.112, 111.344, -15.3, -83.573, 50.748]
  Set speed (120.0 mm/s)
  MoveL 3694 to (500.19, 492.3, 7.5) mm, rotated rx 0 ry 90 rz 0 deg; joints [-11.297, -27.106, 111.303, -15.294, -83.539, 50.756]
  Set speed (1000.0 mm/s)
  MoveL 3695 to (500.24, 492.3, 7.5) mm, rotated rx 0 ry 90 rz 0 deg; joints [-11.297, -27.105, 111.297, -15.293, -83.534, 50.758]
  Set speed (1000.0 mm/s)
  MoveL 3696 to (500.24, 493, 7.5) mm, rotated rx 0 ry 90 rz 0 deg; joints [-11.361, -27.102, 111.28, -15.359, -83.522, 50.768]
  Set speed (1000.0 mm/s)
  MoveL 3697 to (497.06, 492.39, 7.5) mm, rotated rx 0 ry 90 rz 0 deg; joints [-11.364, -27.16, 111.673, -15.352, -83.845, 50.679]
  Set speed (1000.0 mm/s)
  MoveL 3698 to (490.68, 490.68, 7.5) mm, rotated rx 0 ry 90 rz 0 deg; joints [-11.324, -27.271, 112.469, -15.293, -84.505, 50.493]
  Set speed (1000.0 mm/s)
  MoveL 3699 to (490.68, 490.68, 7.6) mm, rotated rx 0 ry 90 rz 0 deg; joints [-11.324, -27.282, 112.475, -15.293, -84.5, 50.495]
  Set speed (30.0 mm/s)
  Call Extruder(0.767)
  MoveL 3700 to (509.32, 509.32, 7.6) mm, rotated rx 0 ry 90 rz 0 deg; joints [-12.669, -26.877, 109.782, -16.719, -82.339, 51.265]
  MoveL 3701 to (509.44, 509.44, 7.6) mm, rotated rx 0 ry 90 rz 0 deg; joints [-12.677, -26.874, 109.764, -16.729, -82.325, 51.27]
  Set speed (120.0 mm/s)
  MoveL 3702 to (508.75, 501.15, 7.6) mm, rotated rx 0 ry 90 rz 0 deg; joints [-11.944, -26.923, 110.064, -15.98, -82.541, 51.112]
  Set speed (30.0 mm/s)
  Call Extruder(0.336)
  MoveL 3703 to (500.58, 509.32, 7.6) mm, rotated rx 0 ry 90 rz 0 deg; joints [-12.847, -27.044, 110.828, -16.867, -83.187, 51.029]
  Set speed (120.0 mm/s)
  MoveL 3704 to (499.42, 509.32, 7.6) mm, rotated rx 0 ry 90 rz 0 deg; joints [-12.872, -27.065, 110.965, -16.887, -83.299, 50.997]
  Set speed (30.0 mm/s)
  Call Extruder(0.360)
  MoveL 3705 to (490.68, 500.58, 7.6) mm, rotated rx 0 ry 90 rz 0 deg; joints [-12.247, -27.249, 112.231, -16.226, -84.319, 50.629]
  Set speed (120.0 mm/s)
  MoveL 3706 to (490.68, 499.42, 7.6) mm, rotated rx 0 ry 90 rz 0 deg; joints [-12.139, -27.253, 112.26, -16.117, -84.341, 50.612]
  Set speed (30.0 mm/s)
  Call Extruder(0.282)
  MoveL 3707 to (497.52, 492.57, 7.6) mm, rotated rx 0 ry 90 rz 0 deg; joints [-11.373, -27.162, 111.619, -15.362, -83.791, 50.695]
  MoveL 3708 to (497.65, 492.45, 7.6) mm, rotated rx 0 ry 90 rz 0 deg; joints [-11.359, -27.16, 111.607, -15.349, -83.781, 50.696]
  Set speed (120.0 mm/s)
  MoveL 3709 to (502.48, 492.58, 7.6) mm, rotated rx 0 ry 90 rz 0 deg; joints [-11.281, -27.074, 111.028, -15.285, -83.304, 50.819]
  Set speed (30.0 mm/s)
  Call Extruder(0.228)
  MoveL 3710 to (508.01, 498.11, 7.6) mm, rotated rx 0 ry 90 rz 0 deg; joints [-11.683, -26.95, 110.23, -15.712, -82.667, 51.044]
  MoveL 3711 to (508.13, 498.23, 7.6) mm, rotated rx 0 ry 90 rz 0 deg; joints [-11.692, -26.947, 110.213, -15.721, -82.653, 51.049]
  Set speed (120.0 mm/s)
  MoveL 3712 to (509.32, 490.68, 7.6) mm, rotated rx 0 ry 90 rz 0 deg; joints [-10.985, -26.954, 110.252, -15.008, -82.662, 50.96]
  Set speed (30.0 mm/s)
  Call Extruder(0.767)
  MoveL 3713 to (490.68, 509.32, 7.6) mm, rotated rx 0 ry 90 rz 0 deg; joints [-13.056, -27.216, 112, -17.045, -84.149, 50.755]
  MoveL 3714 to (490.56, 509.44, 7.6) mm, rotated rx 0 ry 90 rz 0 deg; joints [-13.07, -27.218, 112.011, -17.058, -84.158, 50.754]
  Set speed (120.0 mm/s)
  MoveL 3715 to (499.7, 492.37, 7.6) mm, rotated rx 0 ry 90 rz 0 deg; joints [-11.313, -27.125, 111.364, -15.308, -83.58, 50.747]
  Set speed (1000.0 mm/s)
  MoveL 3716 to (499.77, 492.3, 7.6) mm, rotated rx 0 ry 90 rz 0 deg; joints [-11.305, -27.124, 111.357, -15.301, -83.574, 50.747]
  Set speed (15.0 mm/s)
  Call Extruder(0.010)
  MoveL 3717 to (500.12, 492.3, 7.6) mm, rotated rx 0 ry 90 rz 0 deg; joints [-11.299, -27.117, 111.316, -15.295, -83.54, 50.756]
  Call Extruder(0.000)
  MoveL 3718 to (500.12, 492.3, 7.6) mm, rotated rx 0 ry 90 rz 0 deg; joints [-11.299, -27.117, 111.315, -15.295, -83.54, 50.756]
  Call Extruder(0.062)
  MoveL 3719 to (502.27, 492.3, 7.6) mm, rotated rx 0 ry 90 rz 0 deg; joints [-11.259, -27.079, 111.06, -15.262, -83.329, 50.81]
  Call Extruder(0.055)
  MoveL 3720 to (502.27, 490.4, 7.6) mm, rotated rx 0 ry 90 rz 0 deg; joints [-11.085, -27.086, 111.104, -15.086, -83.361, 50.782]
  Call Extruder(0.213)
  MoveL 3721 to (509.6, 490.4, 7.6) mm, rotated rx 0 ry 90 rz 0 deg; joints [-10.955, -26.949, 110.224, -14.978, -82.639, 50.963]
  Call Extruder(0.232)
  MoveL 3722 to (509.6, 498.39, 7.6) mm, rotated rx 0 ry 90 rz 0 deg; joints [-11.679, -26.918, 110.032, -15.713, -82.506, 51.089]
  Call Extruder(0.056)
  MoveL 3723 to (507.66, 498.39, 7.6) mm, rotated rx 0 ry 90 rz 0 deg; joints [-11.715, -26.956, 110.265, -15.743, -82.696, 51.04]
  Call Extruder(0.072)
  MoveL 3724 to (507.66, 500.87, 7.6) mm, rotated rx 0 ry 90 rz 0 deg; joints [-11.94, -26.946, 110.203, -15.971, -82.653, 51.08]
  Call Extruder(0.056)
  MoveL 3725 to (509.6, 500.87, 7.6) mm, rotated rx 0 ry 90 rz 0 deg; joints [-11.903, -26.908, 109.969, -15.941, -82.463, 51.13]
  Call Extruder(0.254)
  MoveL 3726 to (509.6, 509.6, 7.6) mm, rotated rx 0 ry 90 rz 0 deg; joints [-12.688, -26.871, 109.74, -16.74, -82.307, 51.277]
  Call Extruder(0.559)
  MoveL 3727 to (490.4, 509.6, 7.6) mm, rotated rx 0 ry 90 rz 0 deg; joints [-13.088, -27.22, 112.025, -17.076, -84.17, 50.752]
  MoveL 3728 to (490.4, 490.4, 7.6) mm, rotated rx 0 ry 90 rz 0 deg; joints [-11.303, -27.287, 112.514, -15.271, -84.532, 50.484]
  Call Extruder(0.186)
  MoveL 3729 to (496.79, 490.4, 7.6) mm, rotated rx 0 ry 90 rz 0 deg; joints [-11.185, -27.182, 111.757, -15.17, -83.901, 50.646]
  Call Extruder(0.055)
  MoveL 3730 to (496.79, 492.3, 7.6) mm, rotated rx 0 ry 90 rz 0 deg; joints [-11.36, -27.175, 111.712, -15.347, -83.868, 50.672]
  Call Extruder(0.074)
  MoveL 3731 to (499.35, 492.29, 7.6) mm, rotated rx 0 ry 90 rz 0 deg; joints [-11.313, -27.131, 111.408, -15.307, -83.617, 50.737]
  Call Extruder(0.023)
  MoveL 3732 to (499.35, 491.5, 7.6) mm, rotated rx 0 ry 90 rz 0 deg; joints [-11.239, -27.134, 111.427, -15.233, -83.63, 50.725]
  Call Extruder(0.032)
  MoveL 3733 to (499.34, 490.4, 7.6) mm, rotated rx 0 ry 90 rz 0 deg; joints [-11.138, -27.138, 111.453, -15.13, -83.649, 50.71]
  Call Extruder(0.013)
  MoveL 3734 to (499.78, 490.4, 7.6) mm, rotated rx 0 ry 90 rz 0 deg; joints [-11.13, -27.13, 111.402, -15.124, -83.606, 50.72]
  Call Extruder(0.020)
  MoveL 3735 to (499.78, 491.5, 7.6) mm, rotated rx 0 ry 90 rz 0 deg; joints [-11.231, -27.126, 111.376, -15.226, -83.588, 50.736]
  Call Extruder(0.013)
  MoveL 3736 to (499.78, 491.94, 7.6) mm, rotated rx 0 ry 90 rz 0 deg; joints [-11.273, -27.125, 111.365, -15.268, -83.58, 50.742]
  Call Extruder(0.000)
  MoveL 3737 to (499.77, 491.95, 7.6) mm, rotated rx 0 ry 90 rz 0 deg; joints [-11.273, -27.125, 111.366, -15.268, -83.58, 50.742]
  Call Extruder(0.007)
  MoveL 3738 to (499.77, 492.3, 7.6) mm, rotated rx 0 ry 90 rz 0 deg; joints [-11.305, -27.124, 111.357, -15.301, -83.574, 50.747]
  Set speed (120.0 mm/s)
  MoveL 3739 to (500.12, 492.3, 7.6) mm, rotated rx 0 ry 90 rz 0 deg; joints [-11.299, -27.117, 111.316, -15.295, -83.54, 50.756]
  Set speed (1000.0 mm/s)
  MoveL 3740 to (500.12, 492.3, 7.6) mm, rotated rx 0 ry 90 rz 0 deg; joints [-11.299, -27.117, 111.315, -15.295, -83.54, 50.756]
  Set speed (1000.0 mm/s)
  MoveL 3741 to (500.17, 492.3, 7.6) mm, rotated rx 0 ry 90 rz 0 deg; joints [-11.298, -27.117, 111.31, -15.295, -83.535, 50.758]
  Set speed (1000.0 mm/s)
  MoveL 3742 to (500.17, 493, 7.6) mm, rotated rx 0 ry 90 rz 0 deg; joints [-11.362, -27.114, 111.293, -15.36, -83.523, 50.768]
  Set speed (1000.0 mm/s)
  MoveL 3743 to (497.1, 492.39, 7.6) mm, rotated rx 0 ry 90 rz 0 deg; joints [-11.363, -27.17, 111.673, -15.352, -83.836, 50.681]
  Set speed (1000.0 mm/s)
  MoveL 3744 to (490.68, 490.68, 7.6) mm, rotated rx 0 ry 90 rz 0 deg; joints [-11.324, -27.282, 112.475, -15.293, -84.5, 50.495]
  Set speed (1000.0 mm/s)
  MoveL 3745 to (490.68, 490.68, 7.7) mm, rotated rx 0 ry 90 rz 0 deg; joints [-11.324, -27.293, 112.48, -15.293, -84.495, 50.496]
  Set speed (30.0 mm/s)
  Call Extruder(0.767)
  MoveL 3746 to (509.32, 509.32, 7.7) mm, rotated rx 0 ry 90 rz 0 deg; joints [-12.669, -26.888, 109.787, -16.719, -82.334, 51.266]
  MoveL 3747 to (509.44, 509.44, 7.7) mm, rotated rx 0 ry 90 rz 0 deg; joints [-12.677, -26.885, 109.769, -16.729, -82.32, 51.272]
  Set speed (120.0 mm/s)
  MoveL 3748 to (508.75, 501.15, 7.7) mm, rotated rx 0 ry 90 rz 0 deg; joints [-11.944, -26.934, 110.07, -15.98, -82.536, 51.114]
  Set speed (30.0 mm/s)
  Call Extruder(0.336)
  MoveL 3749 to (500.58, 509.32, 7.7) mm, rotated rx 0 ry 90 rz 0 deg; joints [-12.847, -27.054, 110.833, -16.867, -83.182, 51.03]
  Set speed (120.0 mm/s)
  MoveL 3750 to (499.42, 509.32, 7.7) mm, rotated rx 0 ry 90 rz 0 deg; joints [-12.872, -27.075, 110.971, -16.888, -83.294, 50.999]
  Set speed (30.0 mm/s)
  Call Extruder(0.360)
  MoveL 3751 to (490.68, 500.58, 7.7) mm, rotated rx 0 ry 90 rz 0 deg; joints [-12.247, -27.259, 112.236, -16.226, -84.314, 50.63]
  Set speed (120.0 mm/s)
  MoveL 3752 to (490.68, 499.42, 7.7) mm, rotated rx 0 ry 90 rz 0 deg; joints [-12.139, -27.263, 112.266, -16.117, -84.335, 50.614]
  Set speed (30.0 mm/s)
  Call Extruder(0.282)
  MoveL 3753 to (497.52, 492.58, 7.7) mm, rotated rx 0 ry 90 rz 0 deg; joints [-11.373, -27.173, 111.624, -15.362, -83.786, 50.696]
  MoveL 3754 to (497.65, 492.45, 7.7) mm, rotated rx 0 ry 90 rz 0 deg; joints [-11.359, -27.171, 111.612, -15.349, -83.776, 50.697]
  Set speed (120.0 mm/s)
  MoveL 3755 to (502.48, 492.58, 7.7) mm, rotated rx 0 ry 90 rz 0 deg; joints [-11.281, -27.085, 111.033, -15.285, -83.299, 50.821]
  Set speed (30.0 mm/s)
  Call Extruder(0.228)
  MoveL 3756 to (508.01, 498.11, 7.7) mm, rotated rx 0 ry 90 rz 0 deg; joints [-11.683, -26.961, 110.236, -15.712, -82.662, 51.045]
  MoveL 3757 to (508.13, 498.23, 7.7) mm, rotated rx 0 ry 90 rz 0 deg; joints [-11.692, -26.958, 110.218, -15.721, -82.648, 51.051]
  Set speed (120.0 mm/s)
  MoveL 3758 to (509.32, 490.68, 7.7) mm, rotated rx 0 ry 90 rz 0 deg; joints [-10.985, -26.964, 110.257, -15.008, -82.657, 50.961]
  Set speed (30.0 mm/s)
  Call Extruder(0.767)
  MoveL 3759 to (490.68, 509.32, 7.7) mm, rotated rx 0 ry 90 rz 0 deg; joints [-13.056, -27.227, 112.005, -17.045, -84.144, 50.757]
  MoveL 3760 to (490.56, 509.44, 7.7) mm, rotated rx 0 ry 90 rz 0 deg; joints [-13.07, -27.229, 112.016, -17.058, -84.153, 50.755]
  Set speed (120.0 mm/s)
  MoveL 3761 to (499.64, 492.37, 7.7) mm, rotated rx 0 ry 90 rz 0 deg; joints [-11.314, -27.136, 111.376, -15.309, -83.581, 50.747]
  Set speed (1000.0 mm/s)
  MoveL 3762 to (499.71, 492.3, 7.7) mm, rotated rx 0 ry 90 rz 0 deg; joints [-11.306, -27.135, 111.37, -15.302, -83.575, 50.747]
  Set speed (15.0 mm/s)
  Call Extruder(0.010)
  MoveL 3763 to (500.06, 492.29, 7.7) mm, rotated rx 0 ry 90 rz 0 deg; joints [-11.3, -27.129, 111.328, -15.296, -83.541, 50.756]
  Call Extruder(0.000)
  MoveL 3764 to (500.06, 492.3, 7.7) mm, rotated rx 0 ry 90 rz 0 deg; joints [-11.3, -27.129, 111.328, -15.296, -83.541, 50.756]
  Call Extruder(0.062)
  MoveL 3765 to (502.2, 492.3, 7.7) mm, rotated rx 0 ry 90 rz 0 deg; joints [-11.261, -27.091, 111.072, -15.264, -83.33, 50.81]
  Call Extruder(0.055)
  MoveL 3766 to (502.21, 490.4, 7.7) mm, rotated rx 0 ry 90 rz 0 deg; joints [-11.086, -27.098, 111.117, -15.087, -83.362, 50.782]
  Call Extruder(0.215)
  MoveL 3767 to (509.6, 490.4, 7.7) mm, rotated rx 0 ry 90 rz 0 deg; joints [-10.955, -26.96, 110.23, -14.979, -82.634, 50.964]
  Call Extruder(0.232)
  MoveL 3768 to (509.6, 498.39, 7.7) mm, rotated rx 0 ry 90 rz 0 deg; joints [-11.678, -26.929, 110.037, -15.713, -82.501, 51.09]
  Call Extruder(0.046)
  MoveL 3769 to (508.01, 498.39, 7.7) mm, rotated rx 0 ry 90 rz 0 deg; joints [-11.708, -26.959, 110.228, -15.738, -82.656, 51.05]
  Call Extruder(0.010)
  MoveL 3770 to (507.66, 498.39, 7.7) mm, rotated rx 0 ry 90 rz 0 deg; joints [-11.715, -26.966, 110.27, -15.743, -82.691, 51.041]
  Call Extruder(0.007)
  MoveL 3771 to (507.66, 498.74, 7.7) mm, rotated rx 0 ry 90 rz 0 deg; joints [-11.747, -26.965, 110.261, -15.775, -82.685, 51.047]
  Call Extruder(0.062)
  MoveL 3772 to (507.66, 500.87, 7.7) mm, rotated rx 0 ry 90 rz 0 deg; joints [-11.939, -26.956, 110.208, -15.971, -82.647, 51.081]
  Call Extruder(0.056)
  MoveL 3773 to (509.6, 500.87, 7.7) mm, rotated rx 0 ry 90 rz 0 deg; joints [-11.903, -26.918, 109.975, -15.941, -82.458, 51.131]
  Call Extruder(0.254)
  MoveL 3774 to (509.6, 509.6, 7.7) mm, rotated rx 0 ry 90 rz 0 deg; joints [-12.688, -26.881, 109.746, -16.741, -82.302, 51.279]
  Call Extruder(0.559)
  MoveL 3775 to (490.4, 509.6, 7.7) mm, rotated rx 0 ry 90 rz 0 deg; joints [-13.088, -27.231, 112.03, -17.076, -84.165, 50.753]
  MoveL 3776 to (490.4, 490.4, 7.7) mm, rotated rx 0 ry 90 rz 0 deg; joints [-11.303, -27.298, 112.519, -15.272, -84.527, 50.485]
  Call Extruder(0.188)
  MoveL 3777 to (496.84, 490.4, 7.7) mm, rotated rx 0 ry 90 rz 0 deg; joints [-11.184, -27.192, 111.756, -15.169, -83.891, 50.648]
  Call Extruder(0.055)
  MoveL 3778 to (496.85, 492.3, 7.7) mm, rotated rx 0 ry 90 rz 0 deg; joints [-11.359, -27.185, 111.711, -15.347, -83.858, 50.675]
  Call Extruder(0.074)
  MoveL 3779 to (499.41, 492.29, 7.7) mm, rotated rx 0 ry 90 rz 0 deg; joints [-11.312, -27.141, 111.407, -15.306, -83.606, 50.74]
  Call Extruder(0.022)
  MoveL 3780 to (499.4, 491.54, 7.7) mm, rotated rx 0 ry 90 rz 0 deg; joints [-11.242, -27.143, 111.425, -15.236, -83.619, 50.729]
  Call Extruder(0.033)
  MoveL 3781 to (499.4, 490.4, 7.7) mm, rotated rx 0 ry 90 rz 0 deg; joints [-11.137, -27.147, 111.451, -15.13, -83.638, 50.713]
  Call Extruder(0.009)
  MoveL 3782 to (499.72, 490.4, 7.7) mm, rotated rx 0 ry 90 rz 0 deg; joints [-11.131, -27.142, 111.414, -15.125, -83.607, 50.72]
  Call Extruder(0.015)
  MoveL 3783 to (499.72, 491.53, 7.7) mm, rotated rx 0 ry 90 rz 0 deg; joints [-11.236, -27.138, 111.387, -15.231, -83.588, 50.737]
  Call Extruder(0.012)
  MoveL 3784 to (499.71, 491.94, 7.7) mm, rotated rx 0 ry 90 rz 0 deg; joints [-11.274, -27.137, 111.378, -15.269, -83.581, 50.742]
  Call Extruder(0.000)
  MoveL 3785 to (499.71, 491.94, 7.7) mm, rotated rx 0 ry 90 rz 0 deg; joints [-11.274, -27.137, 111.378, -15.269, -83.581, 50.742]
  Call Extruder(0.007)
  MoveL 3786 to (499.71, 492.3, 7.7) mm, rotated rx 0 ry 90 rz 0 deg; joints [-11.306, -27.135, 111.37, -15.302, -83.575, 50.747]
  Set speed (120.0 mm/s)
  MoveL 3787 to (500.06, 492.29, 7.7) mm, rotated rx 0 ry 90 rz 0 deg; joints [-11.3, -27.129, 111.328, -15.296, -83.541, 50.756]
  Set speed (1000.0 mm/s)
  MoveL 3788 to (500.06, 492.3, 7.7) mm, rotated rx 0 ry 90 rz 0 deg; joints [-11.3, -27.129, 111.328, -15.296, -83.541, 50.756]
  Set speed (1000.0 mm/s)
  MoveL 3789 to (500.11, 492.3, 7.7) mm, rotated rx 0 ry 90 rz 0 deg; joints [-11.299, -27.128, 111.322, -15.296, -83.536, 50.757]
  Set speed (1000.0 mm/s)
  MoveL 3790 to (500.11, 493, 7.7) mm, rotated rx 0 ry 90 rz 0 deg; joints [-11.363, -27.126, 111.305, -15.361, -83.524, 50.768]
  Set speed (1000.0 mm/s)
  MoveL 3791 to (497.15, 492.39, 7.7) mm, rotated rx 0 ry 90 rz 0 deg; joints [-11.363, -27.18, 111.673, -15.351, -83.826, 50.684]
  Set speed (1000.0 mm/s)
  MoveL 3792 to (490.68, 490.68, 7.7) mm, rotated rx 0 ry 90 rz 0 deg; joints [-11.324, -27.293, 112.48, -15.293, -84.495, 50.496]
  Set speed (1000.0 mm/s)
  MoveL 3793 to (490.68, 490.68, 7.8) mm, rotated rx 0 ry 90 rz 0 deg; joints [-11.324, -27.303, 112.485, -15.294, -84.489, 50.498]
  Set speed (30.0 mm/s)
  Call Extruder(0.767)
  MoveL 3794 to (509.32, 509.32, 7.8) mm, rotated rx 0 ry 90 rz 0 deg; joints [-12.669, -26.898, 109.792, -16.72, -82.329, 51.268]
  MoveL 3795 to (509.44, 509.44, 7.8) mm, rotated rx 0 ry 90 rz 0 deg; joints [-12.677, -26.895, 109.774, -16.729, -82.315, 51.273]
  Set speed (120.0 mm/s)
  MoveL 3796 to (508.75, 501.15, 7.8) mm, rotated rx 0 ry 90 rz 0 deg; joints [-11.944, -26.944, 110.075, -15.98, -82.531, 51.115]
  Set speed (30.0 mm/s)
  Call Extruder(0.336)
  MoveL 3797 to (500.58, 509.32, 7.8) mm, rotated rx 0 ry 90 rz 0 deg; joints [-12.847, -27.065, 110.838, -16.868, -83.177, 51.032]
  Set speed (120.0 mm/s)
  MoveL 3798 to (499.42, 509.32, 7.8) mm, rotated rx 0 ry 90 rz 0 deg; joints [-12.872, -27.086, 110.976, -16.888, -83.289, 51]
  Set speed (30.0 mm/s)
  Call Extruder(0.360)
  MoveL 3799 to (490.68, 500.58, 7.8) mm, rotated rx 0 ry 90 rz 0 deg; joints [-12.247, -27.27, 112.241, -16.226, -84.308, 50.632]
  Set speed (120.0 mm/s)
  MoveL 3800 to (490.68, 499.42, 7.8) mm, rotated rx 0 ry 90 rz 0 deg; joints [-12.139, -27.274, 112.271, -16.117, -84.33, 50.615]
  Set speed (30.0 mm/s)
  Call Extruder(0.282)
